KUKA KRL program: EPS_2_26115_ST7258_A_20260223020030.src

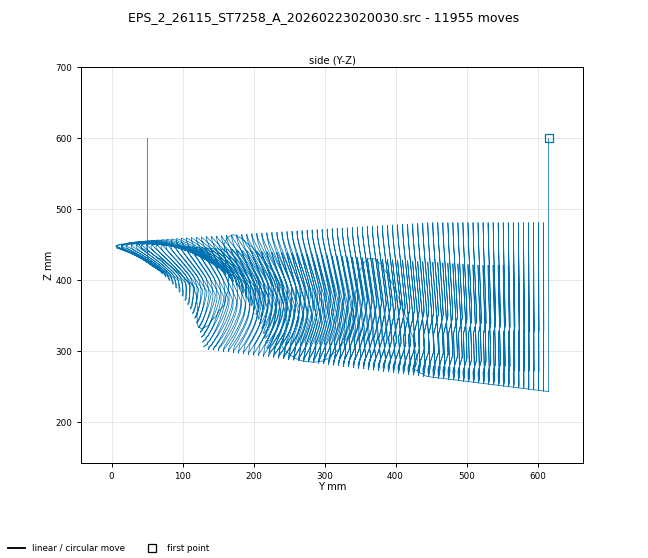
[picture p0: tool path of EPS_2_26115_ST7258_A_20260223020030.src, 11955 of 11957 moves have a stored position in this frame; points joined in program order, loops and branches not executed]
&ACCESS RVP
&REL 4
&COMMENT QRS 19112012
&PARAM EDITMASK = *
DEF PART()
EXT BAS (BAS_COMMAND :IN,REAL :IN )
INT I
BAS (#INITMOV,0 )

;KUKA QRS Post kuka4.cps  Date:22-06-2017 !

File_ID=3071

QRS_PRE_INIT()

;Init var - Until changes are made in qrs_pre_init
Outlet_Square_prg=0
Inlet_1_Square_prg=0
Inlet_2_Square_prg=0
Inlet_3_Square_prg=0
Inlet_4_Square_prg=0
Inlet_5_Square_prg=0

Outlet_1={X 0.000, Y 450.000, Z 332.000, B 0.000, E1 0.000 }
Inlet_1={X 0.000, Y 518.350, Z 272.000, B 0.000, E1 213.000 }
Outlet_1_type=299
Inlet_1_type=299
;QRS#1=Sidecore dimensions
;QRS#2=300-12" PVC SDR 35 Cut Back
;QRS#3=300-12" PVC SDR 35
;QRS#4=
;QRS#5=
;QRS#6=
;QRS#7=
;QRS#8=
;QRS#9=16M PSX
;QRS#10=16M PSX
;QRS#11=
;QRS#12=
;QRS#13=
;QRS#14=
;QRS#15=
;QRS#16=1220x127x762 2,5'
;QRS#17=EPS Height
;QRS#18=481,5
;QRS#19=*
;QRS#20= UPDATED VERSION 22-06-2017
;QRS#21=*
Outlet_Square=0150
Inlet_1_Square=0150
Inlet_2_Square=0
Inlet_3_Square=0
Inlet_4_Square=0
Inlet_5_Square=0
Mill_Square=1
Outlet_Square_Prg=216
Inlet_1_Square_prg=206

QRS_INIT()

$ADVANCE=5

; T1
PTP {E1 173.608,E2 173.608}
PTP {X 0,Y 615.508,A -85,B 0,C 180,E1 173.608,E2 173.608,E3 0,E4 0,E5 0,E6 0}
QRS_SPEED_INIT()
LIN {X 0,Y 615.508,Z 600,A -85,B 0,C 180,E1 173.608,E2 173.608,E3 0,E4 0,E5 0,E6 0} C_VEL
LIN {X 0,Y 615.508,Z 253.5,A -85,B 0,C 180,E1 173.608,E2 173.608} C_VEL
LIN {X 0,Y 615.508,Z 245.325,A -85,B 0,C 180,E1 173.608,E2 173.608} C_VEL
LIN {X 0,Y 615.49,Z 243.325,A -85,B 0,C 180,E1 173.422,E2 173.422} C_VEL
LIN {X 0,Y 615.476,Z 243.325,A -85,B 0,C 180,E1 170.802,E2 170.802} C_VEL
LIN {X 0,Y 615.493,Z 243.324,A -85,B 0,C 180,E1 168.14,E2 168.14} C_VEL
LIN {X 0,Y 615.493,Z 243.322,A -85,B 0,C 180,E1 165.452,E2 165.452} C_VEL
LIN {X 0,Y 615.477,Z 243.325,A -85,B 0,C 180,E1 162.73,E2 162.73} C_VEL
LIN {X 0,Y 615.492,Z 243.326,A -85,B 0,C 180,E1 159.968,E2 159.968} C_VEL
LIN {X 0,Y 615.478,Z 243.325,A -85,B 0,C 180,E1 157.156,E2 157.156} C_VEL
LIN {X 0,Y 615.487,Z 243.323,A -85,B 0,C 180,E1 154.432,E2 154.432} C_VEL
LIN {X 0,Y 615.497,Z 243.325,A -85,B 0,C 180,E1 151.549,E2 151.549} C_VEL
LIN {X 0,Y 615.474,Z 243.325,A -85,B 0,C 180,E1 148.917,E2 148.917} C_VEL
LIN {X 0,Y 615.486,Z 243.326,A -85,B 0,C 180,E1 146.467,E2 146.467} C_VEL
LIN {X 0,Y 615.483,Z 243.324,A -85,B 0,C 180,E1 143.576,E2 143.576} C_VEL
LIN {X 0,Y 615.486,Z 243.325,A -85,B 0,C 180,E1 140.939,E2 140.939} C_VEL
LIN {X 0,Y 615.491,Z 243.326,A -85,B 0,C 180,E1 137.92,E2 137.92} C_VEL
LIN {X 0,Y 615.49,Z 243.326,A -85,B 0,C 180,E1 134.933,E2 134.933} C_VEL
LIN {X 0,Y 615.49,Z 243.322,A -85,B 0,C 180,E1 132.082,E2 132.082} C_VEL
LIN {X 0,Y 615.489,Z 243.325,A -85,B 0,C 180,E1 129.75,E2 129.75} C_VEL
LIN {X 0,Y 615.475,Z 243.325,A -85,B 0,C 180,E1 126.937,E2 126.937} C_VEL
LIN {X 0,Y 615.481,Z 243.325,A -85,B 0,C 180,E1 124.702,E2 124.702} C_VEL
LIN {X 0,Y 615.497,Z 243.325,A -85,B 0,C 180,E1 122.335,E2 122.335} C_VEL
LIN {X 0,Y 615.477,Z 243.326,A -85,B 0,C 180,E1 119.407,E2 119.407} C_VEL
LIN {X 0,Y 615.498,Z 243.325,A -85,B 0,C 180,E1 117.05,E2 117.05} C_VEL
LIN {X 0,Y 615.492,Z 243.326,A -85,B 0,C 180,E1 114.012,E2 114.012} C_VEL
LIN {X 0,Y 615.475,Z 243.325,A -85,B 0,C 180,E1 111.433,E2 111.433} C_VEL
LIN {X 0,Y 615.488,Z 243.326,A -85,B 0,C 180,E1 108.609,E2 108.609} C_VEL
LIN {X 0,Y 615.478,Z 243.325,A -85,B 0,C 180,E1 105.906,E2 105.906} C_VEL
LIN {X 0,Y 615.485,Z 243.324,A -85,B 0,C 180,E1 103.202,E2 103.202} C_VEL
LIN {X 0,Y 615.495,Z 243.323,A -85,B 0,C 180,E1 100.527,E2 100.527} C_VEL
LIN {X 0,Y 615.476,Z 243.325,A -85,B 0,C 180,E1 97.876,E2 97.876} C_VEL
LIN {X 0,Y 615.488,Z 243.326,A -85,B 0,C 180,E1 95.242,E2 95.242} C_VEL
LIN {X 0,Y 615.479,Z 246.1,A -85,B 0,C 180,E1 92.618,E2 92.618} C_VEL
LIN {X 0,Y 615.467,Z 248.837,A -85,B 0,C 180,E1 90,E2 90} C_VEL
LIN {X 0,Y 615.457,Z 251.727,A -85,B 0,C 180,E1 87.382,E2 87.382} C_VEL
LIN {X 0,Y 615.479,Z 254.78,A -85,B 0,C 180,E1 84.759,E2 84.759} C_VEL
LIN {X 0,Y 615.427,Z 257.933,A -85,B 0,C 180,E1 82.124,E2 82.124} C_VEL
LIN {X 0,Y 615.459,Z 261.171,A -85,B 0,C 180,E1 79.473,E2 79.473} C_VEL
LIN {X 0,Y 615.457,Z 264.49,A -85,B 0,C 180,E1 76.799,E2 76.799} C_VEL
LIN {X 0,Y 615.42,Z 267.919,A -85,B 0,C 180,E1 74.094,E2 74.094} C_VEL
LIN {X 0,Y 615.488,Z 268.917,A -85,B 0,C 180,E1 73.307,E2 73.307} C_VEL
LIN {X 0,Y 615.462,Z 288.21,A -85,B 0,C 180,E1 72.943,E2 72.943} C_VEL
LIN {X 0,Y 615.424,Z 303.447,A -85,B 0,C 180,E1 72.514,E2 72.514} C_VEL
LIN {X 0,Y 615.425,Z 318.039,A -85,B 0,C 180,E1 71.961,E2 71.961} C_VEL
LIN {X 0,Y 615.488,Z 332.329,A -85,B 0,C 180,E1 71.268,E2 71.268} C_VEL
LIN {X 0,Y 615.5,Z 345.387,A -85,B 0,C 180,E1 70.49,E2 70.49} C_VEL
LIN {X 0,Y 615.497,Z 358.126,A -85,B 0,C 180,E1 69.57,E2 69.57} C_VEL
LIN {X 0,Y 615.496,Z 369.68,A -85,B 0,C 180,E1 68.569,E2 68.569} C_VEL
LIN {X 0,Y 615.497,Z 379.793,A -85,B 0,C 180,E1 67.526,E2 67.526} C_VEL
LIN {X 0,Y 615.494,Z 388.648,A -85,B 0,C 180,E1 66.445,E2 66.445} C_VEL
LIN {X 0,Y 615.495,Z 397.207,A -85,B 0,C 180,E1 65.189,E2 65.189} C_VEL
LIN {X 0,Y 615.492,Z 404.275,A -85,B 0,C 180,E1 63.921,E2 63.921} C_VEL
LIN {X 0,Y 615.492,Z 409.272,A -85,B 0,C 180,E1 62.824,E2 62.824} C_VEL
LIN {X 0,Y 615.496,Z 413.84,A -85,B 0,C 180,E1 61.546,E2 61.546} C_VEL
LIN {X 0,Y 615.494,Z 417.375,A -85,B 0,C 180,E1 60.202,E2 60.202} C_VEL
LIN {X 0,Y 615.492,Z 419.603,A -85,B 0,C 180,E1 58.911,E2 58.911} C_VEL
LIN {X 0,Y 615.496,Z 420.755,A -85,B 0,C 180,E1 57.544,E2 57.544} C_VEL
LIN {X 0,Y 615.491,Z 420.778,A -85,B 0,C 180,E1 56.463,E2 56.463} C_VEL
LIN {X 0,Y 615.495,Z 419.823,A -85,B 0,C 180,E1 55.186,E2 55.186} C_VEL
LIN {X 0,Y 615.491,Z 418.313,A -85,B 0,C 180,E1 54.164,E2 54.164} C_VEL
LIN {X 0,Y 615.492,Z 415.024,A -85,B 0,C 180,E1 52.759,E2 52.759} C_VEL
LIN {X 0,Y 615.496,Z 410.925,A -85,B 0,C 180,E1 51.516,E2 51.516} C_VEL
LIN {X 0,Y 615.496,Z 405.553,A -85,B 0,C 180,E1 50.251,E2 50.251} C_VEL
LIN {X 0,Y 615.493,Z 398.318,A -85,B 0,C 180,E1 48.903,E2 48.903} C_VEL
LIN {X 0,Y 615.5,Z 390.008,A -85,B 0,C 180,E1 47.649,E2 47.649} C_VEL
LIN {X 0,Y 615.494,Z 381.434,A -85,B 0,C 180,E1 46.568,E2 46.568} C_VEL
LIN {X 0,Y 615.499,Z 370.947,A -85,B 0,C 180,E1 45.461,E2 45.461} C_VEL
LIN {X 0,Y 615.494,Z 359.396,A -85,B 0,C 180,E1 44.441,E2 44.441} C_VEL
LIN {X 0,Y 615.493,Z 346.979,A -85,B 0,C 180,E1 43.525,E2 43.525} C_VEL
LIN {X 0,Y 615.495,Z 333.385,A -85,B 0,C 180,E1 42.699,E2 42.699} C_VEL
LIN {X 0,Y 615.485,Z 321.059,A -85,B 0,C 180,E1 42.081,E2 42.081} C_VEL
LIN {X 0,Y 615.478,Z 306.886,A -85,B 0,C 180,E1 41.511,E2 41.511} C_VEL
LIN {X 0,Y 615.477,Z 291.025,A -85,B 0,C 180,E1 41.033,E2 41.033} C_VEL
LIN {X 0,Y 615.482,Z 275.439,A -85,B 0,C 180,E1 40.712,E2 40.712} C_VEL
LIN {X 0,Y 615.485,Z 268.921,A -85,B 0,C 180,E1 40.605,E2 40.605} C_VEL
LIN {X 0,Y 615.484,Z 265.619,A -85,B 0,C 180,E1 38.013,E2 38.013} C_VEL
LIN {X 0,Y 615.479,Z 262.614,A -85,B 0,C 180,E1 35.615,E2 35.615} C_VEL
LIN {X 0,Y 615.48,Z 259.684,A -85,B 0,C 180,E1 33.235,E2 33.235} C_VEL
LIN {X 0,Y 615.487,Z 256.886,A -85,B 0,C 180,E1 30.918,E2 30.918} C_VEL
LIN {X 0,Y 615.477,Z 253.956,A -85,B 0,C 180,E1 28.45,E2 28.45} C_VEL
LIN {X 0,Y 615.481,Z 250.784,A -85,B 0,C 180,E1 25.715,E2 25.715} C_VEL
LIN {X 0,Y 615.487,Z 248.533,A -85,B 0,C 180,E1 23.555,E2 23.555} C_VEL
LIN {X 0,Y 615.456,Z 246.383,A -85,B 0,C 180,E1 21.432,E2 21.432} C_VEL
LIN {X 0,Y 615.496,Z 243.418,A -85,B 0,C 180,E1 18.609,E2 18.609} C_VEL
LIN {X 0,Y 615.486,Z 243.323,A -85,B 0,C 180,E1 15.904,E2 15.904} C_VEL
LIN {X 0,Y 615.487,Z 243.325,A -85,B 0,C 180,E1 13.2,E2 13.2} C_VEL
LIN {X 0,Y 615.487,Z 243.323,A -85,B 0,C 180,E1 10.526,E2 10.526} C_VEL
LIN {X 0,Y 615.484,Z 243.325,A -85,B 0,C 180,E1 7.875,E2 7.875} C_VEL
LIN {X 0,Y 615.478,Z 243.325,A -85,B 0,C 180,E1 5.241,E2 5.241} C_VEL
LIN {X 0,Y 615.496,Z 243.323,A -85,B 0,C 180,E1 2.617,E2 2.617} C_VEL
LIN {X 0,Y 615.483,Z 243.324,A -85,B 0,C 180,E1 -0.001,E2 -0.001} C_VEL
LIN {X 0,Y 615.49,Z 243.325,A -85,B 0,C 180,E1 -2.619,E2 -2.619} C_VEL
LIN {X 0,Y 615.49,Z 243.322,A -85,B 0,C 180,E1 -5.242,E2 -5.242} C_VEL
LIN {X 0,Y 615.484,Z 243.326,A -85,B 0,C 180,E1 -7.876,E2 -7.876} C_VEL
LIN {X 0,Y 615.474,Z 243.325,A -85,B 0,C 180,E1 -10.528,E2 -10.528} C_VEL
LIN {X 0,Y 615.498,Z 243.323,A -85,B 0,C 180,E1 -13.202,E2 -13.202} C_VEL
LIN {X 0,Y 615.481,Z 243.324,A -85,B 0,C 180,E1 -15.906,E2 -15.906} C_VEL
LIN {X 0,Y 615.48,Z 243.325,A -85,B 0,C 180,E1 -18.647,E2 -18.647} C_VEL
LIN {X 0,Y 615.498,Z 243.324,A -85,B 0,C 180,E1 -21.432,E2 -21.432} C_VEL
LIN {X 0,Y 615.473,Z 243.326,A -85,B 0,C 180,E1 -24.273,E2 -24.273} C_VEL
LIN {X 0,Y 615.498,Z 243.321,A -85,B 0,C 180,E1 -27.048,E2 -27.048} C_VEL
LIN {X 0,Y 615.49,Z 243.325,A -85,B 0,C 180,E1 -29.796,E2 -29.796} C_VEL
LIN {X 0,Y 615.481,Z 243.324,A -85,B 0,C 180,E1 -32.458,E2 -32.458} C_VEL
LIN {X 0,Y 615.493,Z 243.321,A -85,B 0,C 180,E1 -34.815,E2 -34.815} C_VEL
LIN {X 0,Y 615.491,Z 243.325,A -85,B 0,C 180,E1 -37.242,E2 -37.242} C_VEL
LIN {X 0,Y 615.474,Z 243.325,A -85,B 0,C 180,E1 -40.088,E2 -40.088} C_VEL
LIN {X 0,Y 615.481,Z 243.325,A -85,B 0,C 180,E1 -42.354,E2 -42.354} C_VEL
LIN {X 0,Y 615.478,Z 243.325,A -85,B 0,C 180,E1 -45.07,E2 -45.07} C_VEL
LIN {X 0,Y 615.497,Z 243.325,A -85,B 0,C 180,E1 -47.919,E2 -47.919} C_VEL
LIN {X 0,Y 615.498,Z 243.517,A -85,B 0,C 180,E1 -48.717,E2 -48.717} C_VEL
LIN {X 0,Y 615.467,Z 250.403,A -85,B 0,C 180,E1 -51.095,E2 -51.095} C_VEL
LIN {X 0,Y 615.424,Z 257.825,A -85,B 0,C 180,E1 -53.572,E2 -53.572} C_VEL
LIN {X 0,Y 615.43,Z 265.245,A -85,B 0,C 180,E1 -55.975,E2 -55.975} C_VEL
LIN {X 0,Y 615.47,Z 272.654,A -85,B 0,C 180,E1 -58.314,E2 -58.314} C_VEL
LIN {X 0,Y 615.44,Z 281.3,A -85,B 0,C 180,E1 -60.967,E2 -60.967} C_VEL
LIN {X 0,Y 615.44,Z 287.95,A -85,B 0,C 180,E1 -62.964,E2 -62.964} C_VEL
LIN {X 0,Y 615.439,Z 294.876,A -85,B 0,C 180,E1 -65.007,E2 -65.007} C_VEL
LIN {X 0,Y 615.436,Z 302.279,A -85,B 0,C 180,E1 -67.154,E2 -67.154} C_VEL
LIN {X 0,Y 615.448,Z 310.326,A -85,B 0,C 180,E1 -69.453,E2 -69.453} C_VEL
LIN {X 0,Y 615.487,Z 320.751,A -85,B 0,C 180,E1 -72.387,E2 -72.387} C_VEL
LIN {X 0,Y 615.477,Z 325.142,A -85,B 0,C 180,E1 -73.606,E2 -73.606} C_VEL
LIN {X 0,Y 615.494,Z 343.255,A -85,B 0,C 180,E1 -73.9,E2 -73.9} C_VEL
LIN {X 0,Y 615.497,Z 357.822,A -85,B 0,C 180,E1 -74.266,E2 -74.266} C_VEL
LIN {X 0,Y 615.456,Z 372.682,A -85,B 0,C 180,E1 -74.774,E2 -74.774} C_VEL
LIN {X 0,Y 615.465,Z 386.117,A -85,B 0,C 180,E1 -75.366,E2 -75.366} C_VEL
LIN {X 0,Y 615.498,Z 400.019,A -85,B 0,C 180,E1 -76.127,E2 -76.127} C_VEL
LIN {X 0,Y 615.496,Z 412.639,A -85,B 0,C 180,E1 -76.967,E2 -76.967} C_VEL
LIN {X 0,Y 615.496,Z 423.235,A -85,B 0,C 180,E1 -77.805,E2 -77.805} C_VEL
LIN {X 0,Y 615.496,Z 433.979,A -85,B 0,C 180,E1 -78.808,E2 -78.808} C_VEL
LIN {X 0,Y 615.496,Z 444.426,A -85,B 0,C 180,E1 -79.972,E2 -79.972} C_VEL
LIN {X 0,Y 615.495,Z 453.105,A -85,B 0,C 180,E1 -81.133,E2 -81.133} C_VEL
LIN {X 0,Y 615.493,Z 461.227,A -85,B 0,C 180,E1 -82.455,E2 -82.455} C_VEL
LIN {X 0,Y 615.496,Z 467.731,A -85,B 0,C 180,E1 -83.773,E2 -83.773} C_VEL
LIN {X 0,Y 615.496,Z 472.81,A -85,B 0,C 180,E1 -85.088,E2 -85.088} C_VEL
LIN {X 0,Y 615.495,Z 475.741,A -85,B 0,C 180,E1 -86.072,E2 -86.072} C_VEL
LIN {X 0,Y 615.494,Z 478.601,A -85,B 0,C 180,E1 -87.383,E2 -87.383} C_VEL
LIN {X 0,Y 615.492,Z 480.307,A -85,B 0,C 180,E1 -88.692,E2 -88.692} C_VEL
LIN {X 0,Y 615.491,Z 480.889,A -85,B 0,C 180,E1 -90,E2 -90} C_VEL
LIN {X 0,Y 615.492,Z 480.306,A -85,B 0,C 180,E1 -91.309,E2 -91.309} C_VEL
LIN {X 0,Y 615.494,Z 478.599,A -85,B 0,C 180,E1 -92.618,E2 -92.618} C_VEL
LIN {X 0,Y 615.495,Z 475.739,A -85,B 0,C 180,E1 -93.929,E2 -93.929} C_VEL
LIN {X 0,Y 615.491,Z 471.664,A -85,B 0,C 180,E1 -95.242,E2 -95.242} C_VEL
LIN {X 0,Y 615.49,Z 466.16,A -85,B 0,C 180,E1 -96.58,E2 -96.58} C_VEL
LIN {X 0,Y 615.493,Z 459.39,A -85,B 0,C 180,E1 -97.876,E2 -97.876} C_VEL
LIN {X 0,Y 615.495,Z 450.806,A -85,B 0,C 180,E1 -99.199,E2 -99.199} C_VEL
LIN {X 0,Y 615.494,Z 441.663,A -85,B 0,C 180,E1 -100.361,E2 -100.361} C_VEL
LIN {X 0,Y 615.497,Z 432.35,A -85,B 0,C 180,E1 -101.36,E2 -101.36} C_VEL
LIN {X 0,Y 615.496,Z 421.288,A -85,B 0,C 180,E1 -102.363,E2 -102.363} C_VEL
LIN {X 0,Y 615.498,Z 409.147,A -85,B 0,C 180,E1 -103.285,E2 -103.285} C_VEL
LIN {X 0,Y 615.498,Z 396.405,A -85,B 0,C 180,E1 -104.09,E2 -104.09} C_VEL
LIN {X 0,Y 615.456,Z 382.602,A -85,B 0,C 180,E1 -104.804,E2 -104.804} C_VEL
LIN {X 0,Y 615.465,Z 368.172,A -85,B 0,C 180,E1 -105.397,E2 -105.397} C_VEL
LIN {X 0,Y 615.494,Z 353.234,A -85,B 0,C 180,E1 -105.863,E2 -105.863} C_VEL
LIN {X 0,Y 615.493,Z 337.989,A -85,B 0,C 180,E1 -106.198,E2 -106.198} C_VEL
LIN {X 0,Y 615.477,Z 325.142,A -85,B 0,C 180,E1 -106.394,E2 -106.394} C_VEL
LIN {X 0,Y 615.445,Z 315.833,A -85,B 0,C 180,E1 -108.993,E2 -108.993} C_VEL
LIN {X 0,Y 615.497,Z 305.962,A -85,B 0,C 180,E1 -111.784,E2 -111.784} C_VEL
LIN {X 0,Y 615.449,Z 297.34,A -85,B 0,C 180,E1 -114.274,E2 -114.274} C_VEL
LIN {X 0,Y 615.431,Z 289.943,A -85,B 0,C 180,E1 -116.447,E2 -116.447} C_VEL
LIN {X 0,Y 615.422,Z 282.534,A -85,B 0,C 180,E1 -118.662,E2 -118.662} C_VEL
LIN {X 0,Y 615.445,Z 274.614,A -85,B 0,C 180,E1 -121.079,E2 -121.079} C_VEL
LIN {X 0,Y 615.485,Z 266.771,A -85,B 0,C 180,E1 -123.534,E2 -123.534} C_VEL
LIN {X 0,Y 615.446,Z 259.654,A -85,B 0,C 180,E1 -125.828,E2 -125.828} C_VEL
LIN {X 0,Y 615.431,Z 252.875,A -85,B 0,C 180,E1 -128.073,E2 -128.073} C_VEL
LIN {X 0,Y 615.432,Z 246.975,A -85,B 0,C 180,E1 -130.083,E2 -130.083} C_VEL
LIN {X 0,Y 615.495,Z 243.321,A -85,B 0,C 180,E1 -131.379,E2 -131.379} C_VEL
LIN {X 0,Y 615.497,Z 243.325,A -85,B 0,C 180,E1 -134.149,E2 -134.149} C_VEL
LIN {X 0,Y 615.484,Z 243.323,A -85,B 0,C 180,E1 -136.953,E2 -136.953} C_VEL
LIN {X 0,Y 615.492,Z 243.326,A -85,B 0,C 180,E1 -139.394,E2 -139.394} C_VEL
LIN {X 0,Y 615.474,Z 243.325,A -85,B 0,C 180,E1 -141.99,E2 -141.99} C_VEL
LIN {X 0,Y 615.481,Z 243.325,A -85,B 0,C 180,E1 -144.383,E2 -144.383} C_VEL
LIN {X 0,Y 615.492,Z 243.326,A -85,B 0,C 180,E1 -146.764,E2 -146.764} C_VEL
LIN {X 0,Y 615.491,Z 243.323,A -85,B 0,C 180,E1 -149.08,E2 -149.08} C_VEL
LIN {X 0,Y 615.478,Z 243.324,A -85,B 0,C 180,E1 -151.552,E2 -151.552} C_VEL
LIN {X 0,Y 615.486,Z 243.324,A -85,B 0,C 180,E1 -154.284,E2 -154.284} C_VEL
LIN {X 0,Y 615.494,Z 243.326,A -85,B 0,C 180,E1 -157.155,E2 -157.155} C_VEL
LIN {X 0,Y 615.477,Z 243.325,A -85,B 0,C 180,E1 -159.966,E2 -159.966} C_VEL
LIN {X 0,Y 615.496,Z 243.321,A -85,B 0,C 180,E1 -162.729,E2 -162.729} C_VEL
LIN {X 0,Y 615.494,Z 243.324,A -85,B 0,C 180,E1 -165.451,E2 -165.451} C_VEL
LIN {X 0,Y 615.475,Z 243.325,A -85,B 0,C 180,E1 -168.138,E2 -168.138} C_VEL
LIN {X 0,Y 615.497,Z 243.325,A -85,B 0,C 180,E1 -170.801,E2 -170.801} C_VEL
LIN {X 0,Y 615.475,Z 243.325,A -85,B 0,C 180,E1 -173.443,E2 -173.443} C_VEL
LIN {X 0,Y 615.491,Z 243.326,A -85,B 0,C 180,E1 -176.071,E2 -176.071} C_VEL
LIN {X 0,Y 615.493,Z 243.321,A -85,B 0,C 180,E1 -178.691,E2 -178.691} C_VEL
LIN {X 0,Y 615.489,Z 243.326,A -85,B 0,C 180,E1 -181.308,E2 -181.308} C_VEL
LIN {X 0,Y 615.475,Z 243.325,A -85,B 0,C 180,E1 -183.928,E2 -183.928} C_VEL
LIN {X 0,Y 615.49,Z 243.325,A -85,B 0,C 180,E1 -186.578,E2 -186.578} C_VEL
LIN {X 0,Y 614.807,Z 243.471,A -85,B 0,C 180,E1 -187.124,E2 -187.124} C_VEL
LIN {X 0,Y 611.965,Z 243.883,A -85,B 0,C 180,E1 -188.01,E2 -188.01} C_VEL
LIN {X 0,Y 609.573,Z 244.193,A -85,B 0,C 180,E1 -188.722,E2 -188.722} C_VEL
LIN {X 0,Y 608.541,Z 244.311,A -85,B 0,C 180,E1 -189.272,E2 -189.272} C_VEL
LIN {X 0,Y 608.453,Z 244.32,A -85,B 0,C 180,E1 -189.458,E2 -189.458} C_VEL
LIN {X 0,Y 608.468,Z 244.319,A -85,B 0,C 180,E1 -191.999,E2 -191.999} C_VEL
LIN {X 0,Y 608.476,Z 244.319,A -85,B 0,C 180,E1 -194.72,E2 -194.72} C_VEL
LIN {X 0,Y 608.45,Z 244.321,A -85,B 0,C 180,E1 -197.476,E2 -197.476} C_VEL
LIN {X 0,Y 608.461,Z 244.32,A -85,B 0,C 180,E1 -200.273,E2 -200.273} C_VEL
LIN {X 0,Y 608.459,Z 244.32,A -85,B 0,C 180,E1 -202.475,E2 -202.475} C_VEL
LIN {X 0,Y 608.454,Z 244.321,A -85,B 0,C 180,E1 -204.57,E2 -204.57} C_VEL
LIN {X 0,Y 608.474,Z 244.319,A -85,B 0,C 180,E1 -207.206,E2 -207.206} C_VEL
LIN {X 0,Y 608.472,Z 244.318,A -85,B 0,C 180,E1 -209.972,E2 -209.972} C_VEL
LIN {X 0,Y 608.454,Z 244.321,A -85,B 0,C 180,E1 -212.878,E2 -212.878} C_VEL
LIN {X 0,Y 608.446,Z 244.321,A -85,B 0,C 180,E1 -215.276,E2 -215.276} C_VEL
LIN {X 0,Y 608.465,Z 244.319,A -85,B 0,C 180,E1 -218.24,E2 -218.24} C_VEL
LIN {X 0,Y 608.445,Z 244.321,A -85,B 0,C 180,E1 -220.328,E2 -220.328} C_VEL
LIN {X 0,Y 608.453,Z 244.322,A -85,B 0,C 180,E1 -222.958,E2 -222.958} C_VEL
LIN {X 0,Y 608.463,Z 244.319,A -85,B 0,C 180,E1 -225.734,E2 -225.734} C_VEL
LIN {X 0,Y 608.455,Z 244.32,A -85,B 0,C 180,E1 -228.657,E2 -228.657} C_VEL
LIN {X 0,Y 608.463,Z 244.322,A -85,B 0,C 180,E1 -231.411,E2 -231.411} C_VEL
LIN {X 0,Y 608.471,Z 244.318,A -85,B 0,C 180,E1 -233.949,E2 -233.949} C_VEL
LIN {X 0,Y 608.458,Z 244.32,A -85,B 0,C 180,E1 -236.328,E2 -236.328} C_VEL
LIN {X 0,Y 608.472,Z 244.321,A -85,B 0,C 180,E1 -238.726,E2 -238.726} C_VEL
LIN {X 0,Y 608.476,Z 244.317,A -85,B 0,C 180,E1 -241.377,E2 -241.377} C_VEL
LIN {X 0,Y 608.443,Z 244.324,A -85,B 0,C 180,E1 -243.964,E2 -243.964} C_VEL
LIN {X 0,Y 608.467,Z 244.32,A -85,B 0,C 180,E1 -246.155,E2 -246.155} C_VEL
LIN {X 0,Y 608.455,Z 244.321,A -85,B 0,C 180,E1 -249.018,E2 -249.018} C_VEL
LIN {X 0,Y 608.445,Z 244.321,A -85,B 0,C 180,E1 -251.828,E2 -251.828} C_VEL
LIN {X 0,Y 608.467,Z 244.32,A -85,B 0,C 180,E1 -254.594,E2 -254.594} C_VEL
LIN {X 0,Y 608.478,Z 244.318,A -85,B 0,C 180,E1 -257.323,E2 -257.323} C_VEL
LIN {X 0,Y 608.448,Z 244.321,A -85,B 0,C 180,E1 -260.022,E2 -260.022} C_VEL
LIN {X 0,Y 608.481,Z 244.319,A -85,B 0,C 180,E1 -262.7,E2 -262.7} C_VEL
LIN {X 0,Y 608.466,Z 244.32,A -85,B 0,C 180,E1 -264.698,E2 -264.698} C_VEL
LIN {X 0,Y 608.446,Z 246.912,A -85,B 0,C 180,E1 -267.351,E2 -267.351} C_VEL
LIN {X 0,Y 608.416,Z 249.67,A -85,B 0,C 180,E1 -270,E2 -270} C_VEL
LIN {X 0,Y 608.398,Z 252.528,A -85,B 0,C 180,E1 -272.648,E2 -272.648} C_VEL
LIN {X 0,Y 608.436,Z 255.607,A -85,B 0,C 180,E1 -275.302,E2 -275.302} C_VEL
LIN {X 0,Y 608.369,Z 258.782,A -85,B 0,C 180,E1 -277.968,E2 -277.968} C_VEL
LIN {X 0,Y 608.41,Z 262.041,A -85,B 0,C 180,E1 -280.65,E2 -280.65} C_VEL
LIN {X 0,Y 608.392,Z 265.398,A -85,B 0,C 180,E1 -283.358,E2 -283.358} C_VEL
LIN {X 0,Y 608.374,Z 268.851,A -85,B 0,C 180,E1 -286.096,E2 -286.096} C_VEL
LIN {X 0,Y 608.431,Z 269.427,A -85,B 0,C 180,E1 -286.522,E2 -286.522} C_VEL
LIN {X 0,Y 608.668,Z 276.786,A -85,B 0,C 180,E1 -286.637,E2 -286.637} C_VEL
LIN {X 0,Y 608.606,Z 292.383,A -85,B 0,C 180,E1 -286.974,E2 -286.974} C_VEL
LIN {X 0,Y 608.563,Z 307.119,A -85,B 0,C 180,E1 -287.429,E2 -287.429} C_VEL
LIN {X 0,Y 608.534,Z 321.01,A -85,B 0,C 180,E1 -287.995,E2 -287.995} C_VEL
LIN {X 0,Y 608.576,Z 335.698,A -85,B 0,C 180,E1 -288.749,E2 -288.749} C_VEL
LIN {X 0,Y 608.558,Z 348.631,A -85,B 0,C 180,E1 -289.567,E2 -289.567} C_VEL
LIN {X 0,Y 608.52,Z 361.411,A -85,B 0,C 180,E1 -290.54,E2 -290.54} C_VEL
LIN {X 0,Y 608.481,Z 372.102,A -85,B 0,C 180,E1 -291.513,E2 -291.513} C_VEL
LIN {X 0,Y 608.478,Z 381.894,A -85,B 0,C 180,E1 -292.566,E2 -292.566} C_VEL
LIN {X 0,Y 608.479,Z 391.857,A -85,B 0,C 180,E1 -293.844,E2 -293.844} C_VEL
LIN {X 0,Y 608.452,Z 399.992,A -85,B 0,C 180,E1 -295.118,E2 -295.118} C_VEL
LIN {X 0,Y 608.454,Z 406.66,A -85,B 0,C 180,E1 -296.403,E2 -296.403} C_VEL
LIN {X 0,Y 608.434,Z 411.324,A -85,B 0,C 180,E1 -297.518,E2 -297.518} C_VEL
LIN {X 0,Y 608.424,Z 415.044,A -85,B 0,C 180,E1 -298.614,E2 -298.614} C_VEL
LIN {X 0,Y 608.419,Z 418.388,A -85,B 0,C 180,E1 -299.966,E2 -299.966} C_VEL
LIN {X 0,Y 608.413,Z 420.498,A -85,B 0,C 180,E1 -301.319,E2 -301.319} C_VEL
LIN {X 0,Y 608.419,Z 421.382,A -85,B 0,C 180,E1 -302.518,E2 -302.518} C_VEL
LIN {X 0,Y 608.417,Z 421.345,A -85,B 0,C 180,E1 -303.729,E2 -303.729} C_VEL
LIN {X 0,Y 608.419,Z 420.341,A -85,B 0,C 180,E1 -304.904,E2 -304.904} C_VEL
LIN {X 0,Y 608.442,Z 418.457,A -85,B 0,C 180,E1 -306.092,E2 -306.092} C_VEL
LIN {X 0,Y 608.43,Z 415.923,A -85,B 0,C 180,E1 -307.156,E2 -307.156} C_VEL
LIN {X 0,Y 608.427,Z 411.256,A -85,B 0,C 180,E1 -308.59,E2 -308.59} C_VEL
LIN {X 0,Y 608.436,Z 405.765,A -85,B 0,C 180,E1 -309.871,E2 -309.871} C_VEL
LIN {X 0,Y 608.439,Z 398.755,A -85,B 0,C 180,E1 -311.177,E2 -311.177} C_VEL
LIN {X 0,Y 608.473,Z 390.369,A -85,B 0,C 180,E1 -312.449,E2 -312.449} C_VEL
LIN {X 0,Y 608.473,Z 381.58,A -85,B 0,C 180,E1 -313.56,E2 -313.56} C_VEL
LIN {X 0,Y 608.491,Z 371.388,A -85,B 0,C 180,E1 -314.645,E2 -314.645} C_VEL
LIN {X 0,Y 608.507,Z 360.192,A -85,B 0,C 180,E1 -315.649,E2 -315.649} C_VEL
LIN {X 0,Y 608.547,Z 347.477,A -85,B 0,C 180,E1 -316.601,E2 -316.601} C_VEL
LIN {X 0,Y 608.586,Z 334.717,A -85,B 0,C 180,E1 -317.394,E2 -317.394} C_VEL
LIN {X 0,Y 608.597,Z 320.908,A -85,B 0,C 180,E1 -318.098,E2 -318.098} C_VEL
LIN {X 0,Y 608.611,Z 306.371,A -85,B 0,C 180,E1 -318.686,E2 -318.686} C_VEL
LIN {X 0,Y 608.639,Z 290.791,A -85,B 0,C 180,E1 -319.157,E2 -319.157} C_VEL
LIN {X 0,Y 608.672,Z 275.607,A -85,B 0,C 180,E1 -319.473,E2 -319.473} C_VEL
LIN {X 0,Y 608.552,Z 270.28,A -85,B 0,C 180,E1 -319.552,E2 -319.552} C_VEL
LIN {X 0,Y 608.426,Z 269.368,A -85,B 0,C 180,E1 -319.586,E2 -319.586} C_VEL
LIN {X 0,Y 608.413,Z 266,A -85,B 0,C 180,E1 -322.251,E2 -322.251} C_VEL
LIN {X 0,Y 608.408,Z 262.926,A -85,B 0,C 180,E1 -324.721,E2 -324.721} C_VEL
LIN {X 0,Y 608.418,Z 259.991,A -85,B 0,C 180,E1 -327.119,E2 -327.119} C_VEL
LIN {X 0,Y 608.45,Z 256.5,A -85,B 0,C 180,E1 -330.03,E2 -330.03} C_VEL
LIN {X 0,Y 608.431,Z 253.264,A -85,B 0,C 180,E1 -332.8,E2 -332.8} C_VEL
LIN {X 0,Y 608.453,Z 250.402,A -85,B 0,C 180,E1 -335.43,E2 -335.43} C_VEL
LIN {X 0,Y 608.429,Z 247.513,A -85,B 0,C 180,E1 -338.308,E2 -338.308} C_VEL
LIN {X 0,Y 608.434,Z 245.308,A -85,B 0,C 180,E1 -340.43,E2 -340.43} C_VEL
LIN {X 0,Y 608.454,Z 244.4,A -85,B 0,C 180,E1 -341.287,E2 -341.287} C_VEL
LIN {X 0,Y 608.462,Z 244.319,A -85,B 0,C 180,E1 -343.907,E2 -343.907} C_VEL
LIN {X 0,Y 608.463,Z 244.322,A -85,B 0,C 180,E1 -346.644,E2 -346.644} C_VEL
LIN {X 0,Y 608.463,Z 244.319,A -85,B 0,C 180,E1 -349.351,E2 -349.351} C_VEL
LIN {X 0,Y 608.476,Z 244.319,A -85,B 0,C 180,E1 -352.034,E2 -352.034} C_VEL
LIN {X 0,Y 608.459,Z 244.32,A -85,B 0,C 180,E1 -354.699,E2 -354.699} C_VEL
LIN {X 0,Y 608.485,Z 244.318,A -85,B 0,C 180,E1 -357.353,E2 -357.353} C_VEL
LIN {X 0,Y 608.474,Z 244.318,A -85,B 0,C 180,E1 -360.001,E2 -360.001} C_VEL
LIN {X 0,Y 608.48,Z 244.318,A -85,B 0,C 180,E1 -362.649,E2 -362.649} C_VEL
LIN {X 0,Y 608.468,Z 244.319,A -85,B 0,C 180,E1 -365.302,E2 -365.302} C_VEL
LIN {X 0,Y 608.475,Z 244.319,A -85,B 0,C 180,E1 -367.968,E2 -367.968} C_VEL
LIN {X 0,Y 608.458,Z 244.32,A -85,B 0,C 180,E1 -370.651,E2 -370.651} C_VEL
LIN {X 0,Y 608.472,Z 244.318,A -85,B 0,C 180,E1 -373.357,E2 -373.357} C_VEL
LIN {X 0,Y 608.457,Z 244.322,A -85,B 0,C 180,E1 -376.094,E2 -376.094} C_VEL
LIN {X 0,Y 608.454,Z 244.32,A -85,B 0,C 180,E1 -378.87,E2 -378.87} C_VEL
LIN {X 0,Y 608.471,Z 244.319,A -85,B 0,C 180,E1 -381.692,E2 -381.692} C_VEL
LIN {X 0,Y 608.451,Z 244.323,A -85,B 0,C 180,E1 -384.572,E2 -384.572} C_VEL
LIN {X 0,Y 608.485,Z 244.316,A -85,B 0,C 180,E1 -387.21,E2 -387.21} C_VEL
LIN {X 0,Y 608.468,Z 244.321,A -85,B 0,C 180,E1 -389.973,E2 -389.973} C_VEL
LIN {X 0,Y 608.455,Z 244.321,A -85,B 0,C 180,E1 -392.88,E2 -392.88} C_VEL
LIN {X 0,Y 608.437,Z 244.325,A -85,B 0,C 180,E1 -395.278,E2 -395.278} C_VEL
LIN {X 0,Y 608.465,Z 244.319,A -85,B 0,C 180,E1 -397.747,E2 -397.747} C_VEL
LIN {X 0,Y 608.449,Z 244.322,A -85,B 0,C 180,E1 -400.33,E2 -400.33} C_VEL
LIN {X 0,Y 608.47,Z 244.319,A -85,B 0,C 180,E1 -403.31,E2 -403.31} C_VEL
LIN {X 0,Y 608.471,Z 244.319,A -85,B 0,C 180,E1 -406.132,E2 -406.132} C_VEL
LIN {X 0,Y 608.469,Z 244.331,A -85,B 0,C 180,E1 -408.425,E2 -408.425} C_VEL
LIN {X 0,Y 608.524,Z 251.827,A -85,B 0,C 180,E1 -411.056,E2 -411.056} C_VEL
LIN {X 0,Y 608.47,Z 259.071,A -85,B 0,C 180,E1 -413.5,E2 -413.5} C_VEL
LIN {X 0,Y 608.453,Z 265.26,A -85,B 0,C 180,E1 -415.53,E2 -415.53} C_VEL
LIN {X 0,Y 608.446,Z 272.686,A -85,B 0,C 180,E1 -417.905,E2 -417.905} C_VEL
LIN {X 0,Y 608.502,Z 281.351,A -85,B 0,C 180,E1 -420.603,E2 -420.603} C_VEL
LIN {X 0,Y 608.418,Z 290.016,A -85,B 0,C 180,E1 -423.225,E2 -423.225} C_VEL
LIN {X 0,Y 608.418,Z 297.442,A -85,B 0,C 180,E1 -425.428,E2 -425.428} C_VEL
LIN {X 0,Y 608.477,Z 306.107,A -85,B 0,C 180,E1 -427.953,E2 -427.953} C_VEL
LIN {X 0,Y 608.432,Z 316.01,A -85,B 0,C 180,E1 -430.78,E2 -430.78} C_VEL
LIN {X 0,Y 608.433,Z 325.408,A -85,B 0,C 180,E1 -433.421,E2 -433.421} C_VEL
LIN {X 0,Y 608.669,Z 329.645,A -85,B 0,C 180,E1 -433.487,E2 -433.487} C_VEL
LIN {X 0,Y 608.678,Z 344.777,A -85,B 0,C 180,E1 -433.748,E2 -433.748} C_VEL
LIN {X 0,Y 608.642,Z 359.316,A -85,B 0,C 180,E1 -434.127,E2 -434.127} C_VEL
LIN {X 0,Y 608.586,Z 373.804,A -85,B 0,C 180,E1 -434.64,E2 -434.64} C_VEL
LIN {X 0,Y 608.573,Z 387.869,A -85,B 0,C 180,E1 -435.282,E2 -435.282} C_VEL
LIN {X 0,Y 608.562,Z 401.454,A -85,B 0,C 180,E1 -436.05,E2 -436.05} C_VEL
LIN {X 0,Y 608.547,Z 413.86,A -85,B 0,C 180,E1 -436.901,E2 -436.901} C_VEL
LIN {X 0,Y 608.522,Z 425.28,A -85,B 0,C 180,E1 -437.833,E2 -437.833} C_VEL
LIN {X 0,Y 608.492,Z 436.655,A -85,B 0,C 180,E1 -438.937,E2 -438.937} C_VEL
LIN {X 0,Y 608.471,Z 447.374,A -85,B 0,C 180,E1 -440.191,E2 -440.191} C_VEL
LIN {X 0,Y 608.464,Z 455.657,A -85,B 0,C 180,E1 -441.365,E2 -441.365} C_VEL
LIN {X 0,Y 608.456,Z 463.428,A -85,B 0,C 180,E1 -442.701,E2 -442.701} C_VEL
LIN {X 0,Y 608.437,Z 469.61,A -85,B 0,C 180,E1 -444.033,E2 -444.033} C_VEL
LIN {X 0,Y 608.427,Z 474.384,A -85,B 0,C 180,E1 -445.363,E2 -445.363} C_VEL
LIN {X 0,Y 608.421,Z 477.886,A -85,B 0,C 180,E1 -446.689,E2 -446.689} C_VEL
LIN {X 0,Y 608.444,Z 480.192,A -85,B 0,C 180,E1 -448.015,E2 -448.015} C_VEL
LIN {X 0,Y 608.434,Z 481.351,A -85,B 0,C 180,E1 -449.339,E2 -449.339} C_VEL
LIN {X 0,Y 608.434,Z 481.35,A -85,B 0,C 180,E1 -450.662,E2 -450.662} C_VEL
LIN {X 0,Y 608.444,Z 480.191,A -85,B 0,C 180,E1 -451.986,E2 -451.986} C_VEL
LIN {X 0,Y 608.421,Z 477.884,A -85,B 0,C 180,E1 -453.311,E2 -453.311} C_VEL
LIN {X 0,Y 608.427,Z 474.381,A -85,B 0,C 180,E1 -454.638,E2 -454.638} C_VEL
LIN {X 0,Y 608.437,Z 469.606,A -85,B 0,C 180,E1 -455.968,E2 -455.968} C_VEL
LIN {X 0,Y 608.456,Z 463.423,A -85,B 0,C 180,E1 -457.3,E2 -457.3} C_VEL
LIN {X 0,Y 608.464,Z 455.651,A -85,B 0,C 180,E1 -458.636,E2 -458.636} C_VEL
LIN {X 0,Y 608.471,Z 447.367,A -85,B 0,C 180,E1 -459.81,E2 -459.81} C_VEL
LIN {X 0,Y 608.492,Z 436.651,A -85,B 0,C 180,E1 -461.063,E2 -461.063} C_VEL
LIN {X 0,Y 608.522,Z 425.269,A -85,B 0,C 180,E1 -462.168,E2 -462.168} C_VEL
LIN {X 0,Y 608.547,Z 413.847,A -85,B 0,C 180,E1 -463.1,E2 -463.1} C_VEL
LIN {X 0,Y 608.564,Z 401.439,A -85,B 0,C 180,E1 -463.95,E2 -463.95} C_VEL
LIN {X 0,Y 608.573,Z 387.849,A -85,B 0,C 180,E1 -464.718,E2 -464.718} C_VEL
LIN {X 0,Y 608.586,Z 373.779,A -85,B 0,C 180,E1 -465.36,E2 -465.36} C_VEL
LIN {X 0,Y 608.659,Z 358.549,A -85,B 0,C 180,E1 -465.895,E2 -465.895} C_VEL
LIN {X 0,Y 608.689,Z 343.224,A -85,B 0,C 180,E1 -466.286,E2 -466.286} C_VEL
LIN {X 0,Y 608.694,Z 327.951,A -85,B 0,C 180,E1 -466.535,E2 -466.535} C_VEL
LIN {X 0,Y 608.441,Z 325.392,A -85,B 0,C 180,E1 -466.584,E2 -466.584} C_VEL
LIN {X 0,Y 608.433,Z 316.006,A -85,B 0,C 180,E1 -469.221,E2 -469.221} C_VEL
LIN {X 0,Y 608.477,Z 306.104,A -85,B 0,C 180,E1 -472.048,E2 -472.048} C_VEL
LIN {X 0,Y 608.419,Z 297.439,A -85,B 0,C 180,E1 -474.573,E2 -474.573} C_VEL
LIN {X 0,Y 608.418,Z 290.012,A -85,B 0,C 180,E1 -476.776,E2 -476.776} C_VEL
LIN {X 0,Y 608.503,Z 281.348,A -85,B 0,C 180,E1 -479.398,E2 -479.398} C_VEL
LIN {X 0,Y 608.446,Z 272.683,A -85,B 0,C 180,E1 -482.096,E2 -482.096} C_VEL
LIN {X 0,Y 608.454,Z 265.256,A -85,B 0,C 180,E1 -484.471,E2 -484.471} C_VEL
LIN {X 0,Y 608.515,Z 257.829,A -85,B 0,C 180,E1 -486.911,E2 -486.911} C_VEL
LIN {X 0,Y 608.529,Z 249.165,A -85,B 0,C 180,E1 -489.865,E2 -489.865} C_VEL
LIN {X 0,Y 608.47,Z 244.319,A -85,B 0,C 180,E1 -491.6,E2 -491.6} C_VEL
LIN {X 0,Y 608.464,Z 244.321,A -85,B 0,C 180,E1 -494.264,E2 -494.264} C_VEL
LIN {X 0,Y 608.449,Z 244.321,A -85,B 0,C 180,E1 -497.04,E2 -497.04} C_VEL
LIN {X 0,Y 608.457,Z 244.32,A -85,B 0,C 180,E1 -499.697,E2 -499.697} C_VEL
LIN {X 0,Y 608.465,Z 244.319,A -85,B 0,C 180,E1 -502.253,E2 -502.253} C_VEL
LIN {X 0,Y 608.458,Z 244.32,A -85,B 0,C 180,E1 -505.094,E2 -505.094} C_VEL
LIN {X 0,Y 608.468,Z 244.32,A -85,B 0,C 180,E1 -507.905,E2 -507.905} C_VEL
LIN {X 0,Y 608.46,Z 244.32,A -85,B 0,C 180,E1 -510.22,E2 -510.22} C_VEL
LIN {X 0,Y 608.485,Z 244.317,A -85,B 0,C 180,E1 -512.792,E2 -512.792} C_VEL
LIN {X 0,Y 608.454,Z 244.321,A -85,B 0,C 180,E1 -515.429,E2 -515.429} C_VEL
LIN {X 0,Y 608.468,Z 244.321,A -85,B 0,C 180,E1 -518.308,E2 -518.308} C_VEL
LIN {X 0,Y 608.477,Z 244.319,A -85,B 0,C 180,E1 -521.283,E2 -521.283} C_VEL
LIN {X 0,Y 608.455,Z 244.32,A -85,B 0,C 180,E1 -523.906,E2 -523.906} C_VEL
LIN {X 0,Y 608.467,Z 244.321,A -85,B 0,C 180,E1 -526.643,E2 -526.643} C_VEL
LIN {X 0,Y 608.458,Z 244.32,A -85,B 0,C 180,E1 -529.349,E2 -529.349} C_VEL
LIN {X 0,Y 608.477,Z 244.318,A -85,B 0,C 180,E1 -532.032,E2 -532.032} C_VEL
LIN {X 0,Y 608.475,Z 244.318,A -85,B 0,C 180,E1 -534.698,E2 -534.698} C_VEL
LIN {X 0,Y 608.471,Z 244.318,A -85,B 0,C 180,E1 -537.351,E2 -537.351} C_VEL
LIN {X 0,Y 608.476,Z 244.319,A -85,B 0,C 180,E1 -539.999,E2 -539.999} C_VEL
LIN {X 0,Y 608.481,Z 244.317,A -85,B 0,C 180,E1 -542.647,E2 -542.647} C_VEL
LIN {X 0,Y 608.466,Z 244.321,A -85,B 0,C 180,E1 -545.301,E2 -545.301} C_VEL
LIN {X 0,Y 608.477,Z 244.317,A -85,B 0,C 180,E1 -547.966,E2 -547.966} C_VEL
LIN {X 0,Y 608.453,Z 244.32,A -85,B 0,C 180,E1 -549.458,E2 -549.458} C_VEL
LIN {X 0,Y 607.78,Z 244.405,A -85,B 0,C 180,E1 -550.011,E2 -550.011} C_VEL
LIN {X 0,Y 604.931,Z 244.76,A -85,B 0,C 180,E1 -550.908,E2 -550.908} C_VEL
LIN {X 0,Y 602.53,Z 245.06,A -85,B 0,C 180,E1 -551.629,E2 -551.629} C_VEL
LIN {X 0,Y 601.499,Z 245.187,A -85,B 0,C 180,E1 -552.186,E2 -552.186} C_VEL
LIN {X 0,Y 601.414,Z 245.197,A -85,B 0,C 180,E1 -552.374,E2 -552.374} C_VEL
LIN {X 0,Y 601.429,Z 245.197,A -85,B 0,C 180,E1 -554.896,E2 -554.896} C_VEL
LIN {X 0,Y 601.431,Z 245.197,A -85,B 0,C 180,E1 -556.985,E2 -556.985} C_VEL
LIN {X 0,Y 601.404,Z 245.199,A -85,B 0,C 180,E1 -559.808,E2 -559.808} C_VEL
LIN {X 0,Y 601.412,Z 245.197,A -85,B 0,C 180,E1 -562.682,E2 -562.682} C_VEL
LIN {X 0,Y 601.402,Z 245.199,A -85,B 0,C 180,E1 -564.877,E2 -564.877} C_VEL
LIN {X 0,Y 601.424,Z 245.196,A -85,B 0,C 180,E1 -567.866,E2 -567.866} C_VEL
LIN {X 0,Y 601.427,Z 245.196,A -85,B 0,C 180,E1 -570.163,E2 -570.163} C_VEL
LIN {X 0,Y 601.421,Z 245.198,A -85,B 0,C 180,E1 -572.715,E2 -572.715} C_VEL
LIN {X 0,Y 601.413,Z 245.197,A -85,B 0,C 180,E1 -575.114,E2 -575.114} C_VEL
LIN {X 0,Y 601.431,Z 245.195,A -85,B 0,C 180,E1 -577.418,E2 -577.418} C_VEL
LIN {X 0,Y 601.408,Z 245.2,A -85,B 0,C 180,E1 -579.994,E2 -579.994} C_VEL
LIN {X 0,Y 601.408,Z 245.198,A -85,B 0,C 180,E1 -582.669,E2 -582.669} C_VEL
LIN {X 0,Y 601.42,Z 245.197,A -85,B 0,C 180,E1 -585.481,E2 -585.481} C_VEL
LIN {X 0,Y 601.42,Z 245.198,A -85,B 0,C 180,E1 -588.405,E2 -588.405} C_VEL
LIN {X 0,Y 601.428,Z 245.195,A -85,B 0,C 180,E1 -590.874,E2 -590.874} C_VEL
LIN {X 0,Y 601.437,Z 245.195,A -85,B 0,C 180,E1 -593.733,E2 -593.733} C_VEL
LIN {X 0,Y 601.425,Z 245.198,A -85,B 0,C 180,E1 -596.686,E2 -596.686} C_VEL
LIN {X 0,Y 601.428,Z 245.196,A -85,B 0,C 180,E1 -599.058,E2 -599.058} C_VEL
LIN {X 0,Y 601.435,Z 245.194,A -85,B 0,C 180,E1 -601.373,E2 -601.373} C_VEL
LIN {X 0,Y 601.405,Z 245.199,A -85,B 0,C 180,E1 -603.636,E2 -603.636} C_VEL
LIN {X 0,Y 601.419,Z 245.196,A -85,B 0,C 180,E1 -606.589,E2 -606.589} C_VEL
LIN {X 0,Y 601.432,Z 245.196,A -85,B 0,C 180,E1 -609.478,E2 -609.478} C_VEL
LIN {X 0,Y 601.391,Z 245.203,A -85,B 0,C 180,E1 -612.311,E2 -612.311} C_VEL
LIN {X 0,Y 601.41,Z 245.2,A -85,B 0,C 180,E1 -614.408,E2 -614.408} C_VEL
LIN {X 0,Y 601.422,Z 245.196,A -85,B 0,C 180,E1 -617.171,E2 -617.171} C_VEL
LIN {X 0,Y 601.428,Z 245.196,A -85,B 0,C 180,E1 -619.904,E2 -619.904} C_VEL
LIN {X 0,Y 601.448,Z 245.194,A -85,B 0,C 180,E1 -622.615,E2 -622.615} C_VEL
LIN {X 0,Y 601.428,Z 245.196,A -85,B 0,C 180,E1 -624.635,E2 -624.635} C_VEL
LIN {X 0,Y 601.373,Z 245.382,A -85,B 0,C 180,E1 -625.307,E2 -625.307} C_VEL
LIN {X 0,Y 601.408,Z 248.19,A -85,B 0,C 180,E1 -627.99,E2 -627.99} C_VEL
LIN {X 0,Y 601.363,Z 250.956,A -85,B 0,C 180,E1 -630.669,E2 -630.669} C_VEL
LIN {X 0,Y 601.33,Z 253.773,A -85,B 0,C 180,E1 -633.35,E2 -633.35} C_VEL
LIN {X 0,Y 601.293,Z 256.881,A -85,B 0,C 180,E1 -636.038,E2 -636.038} C_VEL
LIN {X 0,Y 601.305,Z 260.076,A -85,B 0,C 180,E1 -638.739,E2 -638.739} C_VEL
LIN {X 0,Y 601.291,Z 263.366,A -85,B 0,C 180,E1 -641.46,E2 -641.46} C_VEL
LIN {X 0,Y 601.283,Z 266.752,A -85,B 0,C 180,E1 -644.208,E2 -644.208} C_VEL
LIN {X 0,Y 601.296,Z 269.388,A -85,B 0,C 180,E1 -646.318,E2 -646.318} C_VEL
LIN {X 0,Y 601.892,Z 273.606,A -85,B 0,C 180,E1 -646.398,E2 -646.398} C_VEL
LIN {X 0,Y 601.829,Z 288.933,A -85,B 0,C 180,E1 -646.702,E2 -646.702} C_VEL
LIN {X 0,Y 601.736,Z 303.002,A -85,B 0,C 180,E1 -647.108,E2 -647.108} C_VEL
LIN {X 0,Y 601.654,Z 317.87,A -85,B 0,C 180,E1 -647.68,E2 -647.68} C_VEL
LIN {X 0,Y 601.656,Z 332.13,A -85,B 0,C 180,E1 -648.384,E2 -648.384} C_VEL
LIN {X 0,Y 601.612,Z 345.262,A -85,B 0,C 180,E1 -649.181,E2 -649.181} C_VEL
LIN {X 0,Y 601.542,Z 357.455,A -85,B 0,C 180,E1 -650.071,E2 -650.071} C_VEL
LIN {X 0,Y 601.504,Z 369.176,A -85,B 0,C 180,E1 -651.095,E2 -651.095} C_VEL
LIN {X 0,Y 601.444,Z 379.236,A -85,B 0,C 180,E1 -652.137,E2 -652.137} C_VEL
LIN {X 0,Y 601.434,Z 388.158,A -85,B 0,C 180,E1 -653.227,E2 -653.227} C_VEL
LIN {X 0,Y 601.396,Z 395.525,A -85,B 0,C 180,E1 -654.287,E2 -654.287} C_VEL
LIN {X 0,Y 601.365,Z 403.216,A -85,B 0,C 180,E1 -655.62,E2 -655.62} C_VEL
LIN {X 0,Y 601.352,Z 408.478,A -85,B 0,C 180,E1 -656.74,E2 -656.74} C_VEL
LIN {X 0,Y 601.349,Z 412.855,A -85,B 0,C 180,E1 -657.87,E2 -657.87} C_VEL
LIN {X 0,Y 601.338,Z 415.629,A -85,B 0,C 180,E1 -658.775,E2 -658.775} C_VEL
LIN {X 0,Y 601.328,Z 418.861,A -85,B 0,C 180,E1 -660.169,E2 -660.169} C_VEL
LIN {X 0,Y 601.318,Z 420.93,A -85,B 0,C 180,E1 -661.731,E2 -661.731} C_VEL
LIN {X 0,Y 601.323,Z 421.427,A -85,B 0,C 180,E1 -662.703,E2 -662.703} C_VEL
LIN {X 0,Y 601.316,Z 421.093,A -85,B 0,C 180,E1 -664.125,E2 -664.125} C_VEL
LIN {X 0,Y 601.316,Z 420.135,A -85,B 0,C 180,E1 -665.103,E2 -665.103} C_VEL
LIN {X 0,Y 601.33,Z 417.475,A -85,B 0,C 180,E1 -666.587,E2 -666.587} C_VEL
LIN {X 0,Y 601.339,Z 414.035,A -85,B 0,C 180,E1 -667.848,E2 -667.848} C_VEL
LIN {X 0,Y 601.344,Z 409.404,A -85,B 0,C 180,E1 -669.131,E2 -669.131} C_VEL
LIN {X 0,Y 601.368,Z 404.186,A -85,B 0,C 180,E1 -670.282,E2 -670.282} C_VEL
LIN {X 0,Y 601.383,Z 396.859,A -85,B 0,C 180,E1 -671.591,E2 -671.591} C_VEL
LIN {X 0,Y 601.42,Z 387.914,A -85,B 0,C 180,E1 -672.897,E2 -672.897} C_VEL
LIN {X 0,Y 601.475,Z 378.423,A -85,B 0,C 180,E1 -674.045,E2 -674.045} C_VEL
LIN {X 0,Y 601.483,Z 367.872,A -85,B 0,C 180,E1 -675.121,E2 -675.121} C_VEL
LIN {X 0,Y 601.543,Z 356.712,A -85,B 0,C 180,E1 -676.079,E2 -676.079} C_VEL
LIN {X 0,Y 601.59,Z 343.856,A -85,B 0,C 180,E1 -677.005,E2 -677.005} C_VEL
LIN {X 0,Y 601.67,Z 330.295,A -85,B 0,C 180,E1 -677.807,E2 -677.807} C_VEL
LIN {X 0,Y 601.718,Z 316.125,A -85,B 0,C 180,E1 -678.485,E2 -678.485} C_VEL
LIN {X 0,Y 601.759,Z 302.769,A -85,B 0,C 180,E1 -678.989,E2 -678.989} C_VEL
LIN {X 0,Y 601.843,Z 287.524,A -85,B 0,C 180,E1 -679.421,E2 -679.421} C_VEL
LIN {X 0,Y 601.766,Z 271.639,A -85,B 0,C 180,E1 -679.724,E2 -679.724} C_VEL
LIN {X 0,Y 601.337,Z 269.386,A -85,B 0,C 180,E1 -679.773,E2 -679.773} C_VEL
LIN {X 0,Y 601.318,Z 265.82,A -85,B 0,C 180,E1 -682.632,E2 -682.632} C_VEL
LIN {X 0,Y 601.351,Z 262.833,A -85,B 0,C 180,E1 -685.065,E2 -685.065} C_VEL
LIN {X 0,Y 601.331,Z 259.921,A -85,B 0,C 180,E1 -687.479,E2 -687.479} C_VEL
LIN {X 0,Y 601.351,Z 257.099,A -85,B 0,C 180,E1 -689.863,E2 -689.863} C_VEL
LIN {X 0,Y 601.341,Z 253.608,A -85,B 0,C 180,E1 -692.885,E2 -692.885} C_VEL
LIN {X 0,Y 601.387,Z 250.78,A -85,B 0,C 180,E1 -695.716,E2 -695.716} C_VEL
LIN {X 0,Y 601.371,Z 247.743,A -85,B 0,C 180,E1 -698.76,E2 -698.76} C_VEL
LIN {X 0,Y 601.392,Z 245.203,A -85,B 0,C 180,E1 -701.186,E2 -701.186} C_VEL
LIN {X 0,Y 601.44,Z 245.195,A -85,B 0,C 180,E1 -703.714,E2 -703.714} C_VEL
LIN {X 0,Y 601.416,Z 245.198,A -85,B 0,C 180,E1 -706.485,E2 -706.485} C_VEL
LIN {X 0,Y 601.417,Z 245.197,A -85,B 0,C 180,E1 -709.225,E2 -709.225} C_VEL
LIN {X 0,Y 601.438,Z 245.197,A -85,B 0,C 180,E1 -711.94,E2 -711.94} C_VEL
LIN {X 0,Y 601.423,Z 245.196,A -85,B 0,C 180,E1 -714.637,E2 -714.637} C_VEL
LIN {X 0,Y 601.448,Z 245.195,A -85,B 0,C 180,E1 -717.322,E2 -717.322} C_VEL
LIN {X 0,Y 601.442,Z 245.194,A -85,B 0,C 180,E1 -720.001,E2 -720.001} C_VEL
LIN {X 0,Y 601.445,Z 245.194,A -85,B 0,C 180,E1 -722.68,E2 -722.68} C_VEL
LIN {X 0,Y 601.43,Z 245.196,A -85,B 0,C 180,E1 -725.365,E2 -725.365} C_VEL
LIN {X 0,Y 601.438,Z 245.195,A -85,B 0,C 180,E1 -728.061,E2 -728.061} C_VEL
LIN {X 0,Y 601.424,Z 245.198,A -85,B 0,C 180,E1 -731.015,E2 -731.015} C_VEL
LIN {X 0,Y 601.423,Z 245.196,A -85,B 0,C 180,E1 -733.516,E2 -733.516} C_VEL
LIN {X 0,Y 601.436,Z 245.196,A -85,B 0,C 180,E1 -736.288,E2 -736.288} C_VEL
LIN {X 0,Y 601.416,Z 245.197,A -85,B 0,C 180,E1 -739.099,E2 -739.099} C_VEL
LIN {X 0,Y 601.41,Z 245.198,A -85,B 0,C 180,E1 -741.24,E2 -741.24} C_VEL
LIN {X 0,Y 601.448,Z 245.193,A -85,B 0,C 180,E1 -744.141,E2 -744.141} C_VEL
LIN {X 0,Y 601.456,Z 245.192,A -85,B 0,C 180,E1 -747.111,E2 -747.111} C_VEL
LIN {X 0,Y 601.42,Z 245.196,A -85,B 0,C 180,E1 -749.393,E2 -749.393} C_VEL
LIN {X 0,Y 601.399,Z 245.2,A -85,B 0,C 180,E1 -751.727,E2 -751.727} C_VEL
LIN {X 0,Y 601.429,Z 245.198,A -85,B 0,C 180,E1 -754.119,E2 -754.119} C_VEL
LIN {X 0,Y 601.436,Z 245.197,A -85,B 0,C 180,E1 -757.383,E2 -757.383} C_VEL
LIN {X 0,Y 601.408,Z 245.198,A -85,B 0,C 180,E1 -759.996,E2 -759.996} C_VEL
LIN {X 0,Y 601.409,Z 245.2,A -85,B 0,C 180,E1 -762.671,E2 -762.671} C_VEL
LIN {X 0,Y 601.424,Z 245.197,A -85,B 0,C 180,E1 -765.483,E2 -765.483} C_VEL
LIN {X 0,Y 601.459,Z 245.294,A -85,B 0,C 180,E1 -768.183,E2 -768.183} C_VEL
LIN {X 0,Y 601.582,Z 248.682,A -85,B 0,C 180,E1 -769.408,E2 -769.408} C_VEL
LIN {X 0,Y 601.551,Z 255.357,A -85,B 0,C 180,E1 -771.743,E2 -771.743} C_VEL
LIN {X 0,Y 601.538,Z 262.784,A -85,B 0,C 180,E1 -774.256,E2 -774.256} C_VEL
LIN {X 0,Y 601.524,Z 270.211,A -85,B 0,C 180,E1 -776.693,E2 -776.693} C_VEL
LIN {X 0,Y 601.491,Z 277.638,A -85,B 0,C 180,E1 -779.063,E2 -779.063} C_VEL
LIN {X 0,Y 601.447,Z 286.302,A -85,B 0,C 180,E1 -781.755,E2 -781.755} C_VEL
LIN {X 0,Y 601.43,Z 296.205,A -85,B 0,C 180,E1 -784.754,E2 -784.754} C_VEL
LIN {X 0,Y 601.4,Z 305.146,A -85,B 0,C 180,E1 -787.398,E2 -787.398} C_VEL
LIN {X 0,Y 601.412,Z 314.772,A -85,B 0,C 180,E1 -790.191,E2 -790.191} C_VEL
LIN {X 0,Y 601.376,Z 323.436,A -85,B 0,C 180,E1 -792.663,E2 -792.663} C_VEL
LIN {X 0,Y 601.368,Z 325.398,A -85,B 0,C 180,E1 -793.217,E2 -793.217} C_VEL
LIN {X 0,Y 601.878,Z 329.927,A -85,B 0,C 180,E1 -793.299,E2 -793.299} C_VEL
LIN {X 0,Y 601.866,Z 344.876,A -85,B 0,C 180,E1 -793.561,E2 -793.561} C_VEL
LIN {X 0,Y 601.805,Z 359.316,A -85,B 0,C 180,E1 -793.942,E2 -793.942} C_VEL
LIN {X 0,Y 601.703,Z 373.805,A -85,B 0,C 180,E1 -794.46,E2 -794.46} C_VEL
LIN {X 0,Y 601.661,Z 387.87,A -85,B 0,C 180,E1 -795.109,E2 -795.109} C_VEL
LIN {X 0,Y 601.613,Z 401.592,A -85,B 0,C 180,E1 -795.894,E2 -795.894} C_VEL
LIN {X 0,Y 601.57,Z 415.02,A -85,B 0,C 180,E1 -796.832,E2 -796.832} C_VEL
LIN {X 0,Y 601.513,Z 427.198,A -85,B 0,C 180,E1 -797.86,E2 -797.86} C_VEL
LIN {X 0,Y 601.437,Z 438.277,A -85,B 0,C 180,E1 -798.983,E2 -798.983} C_VEL
LIN {X 0,Y 601.428,Z 447.374,A -85,B 0,C 180,E1 -800.075,E2 -800.075} C_VEL
LIN {X 0,Y 601.386,Z 455.657,A -85,B 0,C 180,E1 -801.262,E2 -801.262} C_VEL
LIN {X 0,Y 601.365,Z 463.429,A -85,B 0,C 180,E1 -802.614,E2 -802.614} C_VEL
LIN {X 0,Y 601.357,Z 469.609,A -85,B 0,C 180,E1 -803.963,E2 -803.963} C_VEL
LIN {X 0,Y 601.33,Z 474.384,A -85,B 0,C 180,E1 -805.308,E2 -805.308} C_VEL
LIN {X 0,Y 601.337,Z 477.887,A -85,B 0,C 180,E1 -806.65,E2 -806.65} C_VEL
LIN {X 0,Y 601.343,Z 480.192,A -85,B 0,C 180,E1 -807.991,E2 -807.991} C_VEL
LIN {X 0,Y 601.335,Z 481.35,A -85,B 0,C 180,E1 -809.331,E2 -809.331} C_VEL
LIN {X 0,Y 601.335,Z 481.35,A -85,B 0,C 180,E1 -810.67,E2 -810.67} C_VEL
LIN {X 0,Y 601.343,Z 480.191,A -85,B 0,C 180,E1 -812.01,E2 -812.01} C_VEL
LIN {X 0,Y 601.337,Z 477.885,A -85,B 0,C 180,E1 -813.351,E2 -813.351} C_VEL
LIN {X 0,Y 601.33,Z 474.382,A -85,B 0,C 180,E1 -814.693,E2 -814.693} C_VEL
LIN {X 0,Y 601.357,Z 469.606,A -85,B 0,C 180,E1 -816.038,E2 -816.038} C_VEL
LIN {X 0,Y 601.365,Z 463.423,A -85,B 0,C 180,E1 -817.386,E2 -817.386} C_VEL
LIN {X 0,Y 601.386,Z 455.651,A -85,B 0,C 180,E1 -818.739,E2 -818.739} C_VEL
LIN {X 0,Y 601.428,Z 447.367,A -85,B 0,C 180,E1 -819.926,E2 -819.926} C_VEL
LIN {X 0,Y 601.461,Z 436.931,A -85,B 0,C 180,E1 -821.165,E2 -821.165} C_VEL
LIN {X 0,Y 601.514,Z 427.188,A -85,B 0,C 180,E1 -822.141,E2 -822.141} C_VEL
LIN {X 0,Y 601.57,Z 415.008,A -85,B 0,C 180,E1 -823.169,E2 -823.169} C_VEL
LIN {X 0,Y 601.608,Z 403.073,A -85,B 0,C 180,E1 -824.012,E2 -824.012} C_VEL
LIN {X 0,Y 601.674,Z 389.521,A -85,B 0,C 180,E1 -824.805,E2 -824.805} C_VEL
LIN {X 0,Y 601.716,Z 374.835,A -85,B 0,C 180,E1 -825.497,E2 -825.497} C_VEL
LIN {X 0,Y 601.792,Z 360.605,A -85,B 0,C 180,E1 -826.016,E2 -826.016} C_VEL
LIN {X 0,Y 601.838,Z 345.718,A -85,B 0,C 180,E1 -826.42,E2 -826.42} C_VEL
LIN {X 0,Y 601.86,Z 330.419,A -85,B 0,C 180,E1 -826.694,E2 -826.694} C_VEL
LIN {X 0,Y 601.558,Z 326.608,A -85,B 0,C 180,E1 -826.754,E2 -826.754} C_VEL
LIN {X 0,Y 601.371,Z 325.391,A -85,B 0,C 180,E1 -826.784,E2 -826.784} C_VEL
LIN {X 0,Y 601.413,Z 316.006,A -85,B 0,C 180,E1 -829.454,E2 -829.454} C_VEL
LIN {X 0,Y 601.426,Z 306.242,A -85,B 0,C 180,E1 -832.28,E2 -832.28} C_VEL
LIN {X 0,Y 601.394,Z 297.439,A -85,B 0,C 180,E1 -834.879,E2 -834.879} C_VEL
LIN {X 0,Y 601.444,Z 289.172,A -85,B 0,C 180,E1 -837.367,E2 -837.367} C_VEL
LIN {X 0,Y 601.449,Z 280.11,A -85,B 0,C 180,E1 -840.163,E2 -840.163} C_VEL
LIN {X 0,Y 601.449,Z 272.683,A -85,B 0,C 180,E1 -842.515,E2 -842.515} C_VEL
LIN {X 0,Y 601.544,Z 264.626,A -85,B 0,C 180,E1 -845.132,E2 -845.132} C_VEL
LIN {X 0,Y 601.579,Z 256.592,A -85,B 0,C 180,E1 -847.832,E2 -847.832} C_VEL
LIN {X 0,Y 601.585,Z 248.681,A -85,B 0,C 180,E1 -850.592,E2 -850.592} C_VEL
LIN {X 0,Y 601.424,Z 245.197,A -85,B 0,C 180,E1 -851.878,E2 -851.878} C_VEL
LIN {X 0,Y 601.429,Z 245.196,A -85,B 0,C 180,E1 -854.535,E2 -854.535} C_VEL
LIN {X 0,Y 601.411,Z 245.2,A -85,B 0,C 180,E1 -857.41,E2 -857.41} C_VEL
LIN {X 0,Y 601.406,Z 245.198,A -85,B 0,C 180,E1 -860.004,E2 -860.004} C_VEL
LIN {X 0,Y 601.441,Z 245.196,A -85,B 0,C 180,E1 -862.618,E2 -862.618} C_VEL
LIN {X 0,Y 601.418,Z 245.197,A -85,B 0,C 180,E1 -865.068,E2 -865.068} C_VEL
LIN {X 0,Y 601.434,Z 245.195,A -85,B 0,C 180,E1 -867.484,E2 -867.484} C_VEL
LIN {X 0,Y 601.433,Z 245.197,A -85,B 0,C 180,E1 -869.851,E2 -869.851} C_VEL
LIN {X 0,Y 601.456,Z 245.194,A -85,B 0,C 180,E1 -872.889,E2 -872.889} C_VEL
LIN {X 0,Y 601.453,Z 245.193,A -85,B 0,C 180,E1 -875.859,E2 -875.859} C_VEL
LIN {X 0,Y 601.411,Z 245.197,A -85,B 0,C 180,E1 -878.76,E2 -878.76} C_VEL
LIN {X 0,Y 601.421,Z 245.197,A -85,B 0,C 180,E1 -881.608,E2 -881.608} C_VEL
LIN {X 0,Y 601.415,Z 245.199,A -85,B 0,C 180,E1 -884.408,E2 -884.408} C_VEL
LIN {X 0,Y 601.422,Z 245.196,A -85,B 0,C 180,E1 -887.171,E2 -887.171} C_VEL
LIN {X 0,Y 601.429,Z 245.197,A -85,B 0,C 180,E1 -889.904,E2 -889.904} C_VEL
LIN {X 0,Y 601.447,Z 245.194,A -85,B 0,C 180,E1 -892.614,E2 -892.614} C_VEL
LIN {X 0,Y 601.416,Z 245.197,A -85,B 0,C 180,E1 -895.307,E2 -895.307} C_VEL
LIN {X 0,Y 601.433,Z 245.197,A -85,B 0,C 180,E1 -897.99,E2 -897.99} C_VEL
LIN {X 0,Y 601.454,Z 245.192,A -85,B 0,C 180,E1 -900.669,E2 -900.669} C_VEL
LIN {X 0,Y 601.43,Z 245.198,A -85,B 0,C 180,E1 -903.349,E2 -903.349} C_VEL
LIN {X 0,Y 601.408,Z 245.198,A -85,B 0,C 180,E1 -906.036,E2 -906.036} C_VEL
LIN {X 0,Y 601.419,Z 245.198,A -85,B 0,C 180,E1 -908.737,E2 -908.737} C_VEL
LIN {X 0,Y 601.417,Z 245.198,A -85,B 0,C 180,E1 -911.458,E2 -911.458} C_VEL
LIN {X 0,Y 601.414,Z 245.197,A -85,B 0,C 180,E1 -912.374,E2 -912.374} C_VEL
LIN {X 0,Y 600.747,Z 245.282,A -85,B 0,C 180,E1 -912.933,E2 -912.933} C_VEL
LIN {X 0,Y 597.895,Z 245.638,A -85,B 0,C 180,E1 -913.841,E2 -913.841} C_VEL
LIN {X 0,Y 595.484,Z 245.937,A -85,B 0,C 180,E1 -914.571,E2 -914.571} C_VEL
LIN {X 0,Y 594.446,Z 246.066,A -85,B 0,C 180,E1 -915.135,E2 -915.135} C_VEL
LIN {X 0,Y 594.36,Z 246.075,A -85,B 0,C 180,E1 -915.326,E2 -915.326} C_VEL
LIN {X 0,Y 594.38,Z 246.076,A -85,B 0,C 180,E1 -917.903,E2 -917.903} C_VEL
LIN {X 0,Y 594.374,Z 246.075,A -85,B 0,C 180,E1 -920.914,E2 -920.914} C_VEL
LIN {X 0,Y 594.391,Z 246.072,A -85,B 0,C 180,E1 -923.703,E2 -923.703} C_VEL
LIN {X 0,Y 594.382,Z 246.073,A -85,B 0,C 180,E1 -926.698,E2 -926.698} C_VEL
LIN {X 0,Y 594.382,Z 246.073,A -85,B 0,C 180,E1 -928.997,E2 -928.997} C_VEL
LIN {X 0,Y 594.384,Z 246.075,A -85,B 0,C 180,E1 -931.643,E2 -931.643} C_VEL
LIN {X 0,Y 594.395,Z 246.073,A -85,B 0,C 180,E1 -934.578,E2 -934.578} C_VEL
LIN {X 0,Y 594.382,Z 246.073,A -85,B 0,C 180,E1 -937.085,E2 -937.085} C_VEL
LIN {X 0,Y 594.373,Z 246.076,A -85,B 0,C 180,E1 -939.773,E2 -939.773} C_VEL
LIN {X 0,Y 594.366,Z 246.075,A -85,B 0,C 180,E1 -942.374,E2 -942.374} C_VEL
LIN {X 0,Y 594.358,Z 246.079,A -85,B 0,C 180,E1 -945.19,E2 -945.19} C_VEL
LIN {X 0,Y 594.383,Z 246.073,A -85,B 0,C 180,E1 -947.625,E2 -947.625} C_VEL
LIN {X 0,Y 594.388,Z 246.075,A -85,B 0,C 180,E1 -950.32,E2 -950.32} C_VEL
LIN {X 0,Y 594.379,Z 246.073,A -85,B 0,C 180,E1 -952.912,E2 -952.912} C_VEL
LIN {X 0,Y 594.376,Z 246.075,A -85,B 0,C 180,E1 -955.86,E2 -955.86} C_VEL
LIN {X 0,Y 594.386,Z 246.075,A -85,B 0,C 180,E1 -958.65,E2 -958.65} C_VEL
LIN {X 0,Y 594.38,Z 246.074,A -85,B 0,C 180,E1 -961.04,E2 -961.04} C_VEL
LIN {X 0,Y 594.381,Z 246.076,A -85,B 0,C 180,E1 -963.975,E2 -963.975} C_VEL
LIN {X 0,Y 594.39,Z 246.073,A -85,B 0,C 180,E1 -966.296,E2 -966.296} C_VEL
LIN {X 0,Y 594.403,Z 246.073,A -85,B 0,C 180,E1 -969.224,E2 -969.224} C_VEL
LIN {X 0,Y 594.373,Z 246.075,A -85,B 0,C 180,E1 -972.095,E2 -972.095} C_VEL
LIN {X 0,Y 594.363,Z 246.077,A -85,B 0,C 180,E1 -974.219,E2 -974.219} C_VEL
LIN {X 0,Y 594.368,Z 246.075,A -85,B 0,C 180,E1 -977.017,E2 -977.017} C_VEL
LIN {X 0,Y 594.39,Z 246.073,A -85,B 0,C 180,E1 -979.784,E2 -979.784} C_VEL
LIN {X 0,Y 594.411,Z 246.07,A -85,B 0,C 180,E1 -982.527,E2 -982.527} C_VEL
LIN {X 0,Y 594.315,Z 246.084,A -85,B 0,C 180,E1 -985.251,E2 -985.251} C_VEL
LIN {X 0,Y 594.354,Z 248.765,A -85,B 0,C 180,E1 -987.967,E2 -987.967} C_VEL
LIN {X 0,Y 594.311,Z 251.551,A -85,B 0,C 180,E1 -990.677,E2 -990.677} C_VEL
LIN {X 0,Y 594.246,Z 254.346,A -85,B 0,C 180,E1 -993.39,E2 -993.39} C_VEL
LIN {X 0,Y 594.25,Z 256.579,A -85,B 0,C 180,E1 -995.429,E2 -995.429} C_VEL
LIN {X 0,Y 594.218,Z 259.757,A -85,B 0,C 180,E1 -998.159,E2 -998.159} C_VEL
LIN {X 0,Y 594.232,Z 263.14,A -85,B 0,C 180,E1 -1001.003,E2 -1001.003} C_VEL
LIN {X 0,Y 594.217,Z 266.92,A -85,B 0,C 180,E1 -1004.113,E2 -1004.113} C_VEL
LIN {X 0,Y 594.215,Z 269.412,A -85,B 0,C 180,E1 -1006.115,E2 -1006.115} C_VEL
LIN {X 0,Y 595.08,Z 273.55,A -85,B 0,C 180,E1 -1006.201,E2 -1006.201} C_VEL
LIN {X 0,Y 595.011,Z 288.94,A -85,B 0,C 180,E1 -1006.509,E2 -1006.509} C_VEL
LIN {X 0,Y 594.911,Z 302.083,A -85,B 0,C 180,E1 -1006.889,E2 -1006.889} C_VEL
LIN {X 0,Y 594.795,Z 316.712,A -85,B 0,C 180,E1 -1007.447,E2 -1007.447} C_VEL
LIN {X 0,Y 594.766,Z 329.608,A -85,B 0,C 180,E1 -1008.07,E2 -1008.07} C_VEL
LIN {X 0,Y 594.671,Z 343.571,A -85,B 0,C 180,E1 -1008.9,E2 -1008.9} C_VEL
LIN {X 0,Y 594.573,Z 355.736,A -85,B 0,C 180,E1 -1009.776,E2 -1009.776} C_VEL
LIN {X 0,Y 594.525,Z 367.305,A -85,B 0,C 180,E1 -1010.771,E2 -1010.771} C_VEL
LIN {X 0,Y 594.426,Z 378.01,A -85,B 0,C 180,E1 -1011.865,E2 -1011.865} C_VEL
LIN {X 0,Y 594.377,Z 387.101,A -85,B 0,C 180,E1 -1012.966,E2 -1012.966} C_VEL
LIN {X 0,Y 594.337,Z 395.92,A -85,B 0,C 180,E1 -1014.243,E2 -1014.243} C_VEL
LIN {X 0,Y 594.302,Z 403.425,A -85,B 0,C 180,E1 -1015.571,E2 -1015.571} C_VEL
LIN {X 0,Y 594.282,Z 408.642,A -85,B 0,C 180,E1 -1016.704,E2 -1016.704} C_VEL
LIN {X 0,Y 594.258,Z 412.986,A -85,B 0,C 180,E1 -1017.848,E2 -1017.848} C_VEL
LIN {X 0,Y 594.245,Z 416.365,A -85,B 0,C 180,E1 -1019.005,E2 -1019.005} C_VEL
LIN {X 0,Y 594.224,Z 419.137,A -85,B 0,C 180,E1 -1020.304,E2 -1020.304} C_VEL
LIN {X 0,Y 594.218,Z 420.863,A -85,B 0,C 180,E1 -1021.62,E2 -1021.62} C_VEL
LIN {X 0,Y 594.236,Z 421.486,A -85,B 0,C 180,E1 -1022.958,E2 -1022.958} C_VEL
LIN {X 0,Y 594.24,Z 421.106,A -85,B 0,C 180,E1 -1024.121,E2 -1024.121} C_VEL
LIN {X 0,Y 594.22,Z 419.737,A -85,B 0,C 180,E1 -1025.417,E2 -1025.417} C_VEL
LIN {X 0,Y 594.229,Z 417.824,A -85,B 0,C 180,E1 -1026.465,E2 -1026.465} C_VEL
LIN {X 0,Y 594.263,Z 413.899,A -85,B 0,C 180,E1 -1027.949,E2 -1027.949} C_VEL
LIN {X 0,Y 594.257,Z 409.21,A -85,B 0,C 180,E1 -1029.25,E2 -1029.25} C_VEL
LIN {X 0,Y 594.272,Z 403.137,A -85,B 0,C 180,E1 -1030.574,E2 -1030.574} C_VEL
LIN {X 0,Y 594.306,Z 395.955,A -85,B 0,C 180,E1 -1031.842,E2 -1031.842} C_VEL
LIN {X 0,Y 594.373,Z 387.678,A -85,B 0,C 180,E1 -1033.048,E2 -1033.048} C_VEL
LIN {X 0,Y 594.445,Z 377.969,A -85,B 0,C 180,E1 -1034.229,E2 -1034.229} C_VEL
LIN {X 0,Y 594.505,Z 367.199,A -85,B 0,C 180,E1 -1035.33,E2 -1035.33} C_VEL
LIN {X 0,Y 594.595,Z 356.103,A -85,B 0,C 180,E1 -1036.283,E2 -1036.283} C_VEL
LIN {X 0,Y 594.674,Z 342.72,A -85,B 0,C 180,E1 -1037.247,E2 -1037.247} C_VEL
LIN {X 0,Y 594.77,Z 329.699,A -85,B 0,C 180,E1 -1038.015,E2 -1038.015} C_VEL
LIN {X 0,Y 594.86,Z 316.375,A -85,B 0,C 180,E1 -1038.657,E2 -1038.657} C_VEL
LIN {X 0,Y 594.94,Z 301.883,A -85,B 0,C 180,E1 -1039.207,E2 -1039.207} C_VEL
LIN {X 0,Y 595.024,Z 286.555,A -85,B 0,C 180,E1 -1039.638,E2 -1039.638} C_VEL
LIN {X 0,Y 595.036,Z 273.169,A -85,B 0,C 180,E1 -1039.896,E2 -1039.896} C_VEL
LIN {X 0,Y 594.238,Z 269.367,A -85,B 0,C 180,E1 -1039.993,E2 -1039.993} C_VEL
LIN {X 0,Y 594.215,Z 265.788,A -85,B 0,C 180,E1 -1042.902,E2 -1042.902} C_VEL
LIN {X 0,Y 594.239,Z 262.188,A -85,B 0,C 180,E1 -1045.881,E2 -1045.881} C_VEL
LIN {X 0,Y 594.276,Z 258.915,A -85,B 0,C 180,E1 -1048.646,E2 -1048.646} C_VEL
LIN {X 0,Y 594.248,Z 256.116,A -85,B 0,C 180,E1 -1051.065,E2 -1051.065} C_VEL
LIN {X 0,Y 594.265,Z 253.842,A -85,B 0,C 180,E1 -1053.296,E2 -1053.296} C_VEL
LIN {X 0,Y 594.325,Z 251.586,A -85,B 0,C 180,E1 -1055.578,E2 -1055.578} C_VEL
LIN {X 0,Y 594.286,Z 248.676,A -85,B 0,C 180,E1 -1058.495,E2 -1058.495} C_VEL
LIN {X 0,Y 594.328,Z 246.083,A -85,B 0,C 180,E1 -1061.085,E2 -1061.085} C_VEL
LIN {X 0,Y 594.409,Z 246.073,A -85,B 0,C 180,E1 -1063.516,E2 -1063.516} C_VEL
LIN {X 0,Y 594.379,Z 246.074,A -85,B 0,C 180,E1 -1066.322,E2 -1066.322} C_VEL
LIN {X 0,Y 594.374,Z 246.074,A -85,B 0,C 180,E1 -1069.096,E2 -1069.096} C_VEL
LIN {X 0,Y 594.414,Z 246.071,A -85,B 0,C 180,E1 -1071.844,E2 -1071.844} C_VEL
LIN {X 0,Y 594.388,Z 246.072,A -85,B 0,C 180,E1 -1074.573,E2 -1074.573} C_VEL
LIN {X 0,Y 594.413,Z 246.071,A -85,B 0,C 180,E1 -1077.29,E2 -1077.29} C_VEL
LIN {X 0,Y 594.411,Z 246.069,A -85,B 0,C 180,E1 -1080.001,E2 -1080.001} C_VEL
LIN {X 0,Y 594.41,Z 246.07,A -85,B 0,C 180,E1 -1082.711,E2 -1082.711} C_VEL
LIN {X 0,Y 594.393,Z 246.073,A -85,B 0,C 180,E1 -1085.428,E2 -1085.428} C_VEL
LIN {X 0,Y 594.414,Z 246.069,A -85,B 0,C 180,E1 -1088.157,E2 -1088.157} C_VEL
LIN {X 0,Y 594.388,Z 246.074,A -85,B 0,C 180,E1 -1091.076,E2 -1091.076} C_VEL
LIN {X 0,Y 594.385,Z 246.073,A -85,B 0,C 180,E1 -1093.679,E2 -1093.679} C_VEL
LIN {X 0,Y 594.392,Z 246.071,A -85,B 0,C 180,E1 -1096.721,E2 -1096.721} C_VEL
LIN {X 0,Y 594.366,Z 246.077,A -85,B 0,C 180,E1 -1099.335,E2 -1099.335} C_VEL
LIN {X 0,Y 594.369,Z 246.077,A -85,B 0,C 180,E1 -1101.504,E2 -1101.504} C_VEL
LIN {X 0,Y 594.386,Z 246.074,A -85,B 0,C 180,E1 -1104.447,E2 -1104.447} C_VEL
LIN {X 0,Y 594.388,Z 246.075,A -85,B 0,C 180,E1 -1106.7,E2 -1106.7} C_VEL
LIN {X 0,Y 594.379,Z 246.076,A -85,B 0,C 180,E1 -1108.999,E2 -1108.999} C_VEL
LIN {X 0,Y 594.375,Z 246.075,A -85,B 0,C 180,E1 -1111.643,E2 -1111.643} C_VEL
LIN {X 0,Y 594.383,Z 246.074,A -85,B 0,C 180,E1 -1114.58,E2 -1114.58} C_VEL
LIN {X 0,Y 594.389,Z 246.073,A -85,B 0,C 180,E1 -1117.609,E2 -1117.609} C_VEL
LIN {X 0,Y 594.37,Z 246.077,A -85,B 0,C 180,E1 -1120.567,E2 -1120.567} C_VEL
LIN {X 0,Y 594.364,Z 246.076,A -85,B 0,C 180,E1 -1123.3,E2 -1123.3} C_VEL
LIN {X 0,Y 594.381,Z 246.074,A -85,B 0,C 180,E1 -1126.159,E2 -1126.159} C_VEL
LIN {X 0,Y 594.426,Z 246.204,A -85,B 0,C 180,E1 -1127.92,E2 -1127.92} C_VEL
LIN {X 0,Y 594.691,Z 249.527,A -85,B 0,C 180,E1 -1129.143,E2 -1129.143} C_VEL
LIN {X 0,Y 594.626,Z 256.666,A -85,B 0,C 180,E1 -1131.672,E2 -1131.672} C_VEL
LIN {X 0,Y 594.585,Z 264.022,A -85,B 0,C 180,E1 -1134.191,E2 -1134.191} C_VEL
LIN {X 0,Y 594.543,Z 271.449,A -85,B 0,C 180,E1 -1136.656,E2 -1136.656} C_VEL
LIN {X 0,Y 594.502,Z 278.875,A -85,B 0,C 180,E1 -1139.054,E2 -1139.054} C_VEL
LIN {X 0,Y 594.457,Z 287.54,A -85,B 0,C 180,E1 -1141.778,E2 -1141.778} C_VEL
LIN {X 0,Y 594.435,Z 296.205,A -85,B 0,C 180,E1 -1144.435,E2 -1144.435} C_VEL
LIN {X 0,Y 594.357,Z 305.657,A -85,B 0,C 180,E1 -1147.267,E2 -1147.267} C_VEL
LIN {X 0,Y 594.357,Z 314.772,A -85,B 0,C 180,E1 -1149.946,E2 -1149.946} C_VEL
LIN {X 0,Y 594.303,Z 324.674,A -85,B 0,C 180,E1 -1152.805,E2 -1152.805} C_VEL
LIN {X 0,Y 594.307,Z 325.419,A -85,B 0,C 180,E1 -1153.018,E2 -1153.018} C_VEL
LIN {X 0,Y 595.081,Z 329.893,A -85,B 0,C 180,E1 -1153.102,E2 -1153.102} C_VEL
LIN {X 0,Y 595.061,Z 345.242,A -85,B 0,C 180,E1 -1153.376,E2 -1153.376} C_VEL
LIN {X 0,Y 594.986,Z 359.315,A -85,B 0,C 180,E1 -1153.752,E2 -1153.752} C_VEL
LIN {X 0,Y 594.861,Z 373.805,A -85,B 0,C 180,E1 -1154.277,E2 -1154.277} C_VEL
LIN {X 0,Y 594.759,Z 387.872,A -85,B 0,C 180,E1 -1154.933,E2 -1154.933} C_VEL
LIN {X 0,Y 594.682,Z 401.414,A -85,B 0,C 180,E1 -1155.715,E2 -1155.715} C_VEL
LIN {X 0,Y 594.587,Z 413.861,A -85,B 0,C 180,E1 -1156.588,E2 -1156.588} C_VEL
LIN {X 0,Y 594.535,Z 425.281,A -85,B 0,C 180,E1 -1157.542,E2 -1157.542} C_VEL
LIN {X 0,Y 594.434,Z 435.715,A -85,B 0,C 180,E1 -1158.572,E2 -1158.572} C_VEL
LIN {X 0,Y 594.38,Z 446.024,A -85,B 0,C 180,E1 -1159.784,E2 -1159.784} C_VEL
LIN {X 0,Y 594.337,Z 454.536,A -85,B 0,C 180,E1 -1160.986,E2 -1160.986} C_VEL
LIN {X 0,Y 594.31,Z 461.614,A -85,B 0,C 180,E1 -1162.184,E2 -1162.184} C_VEL
LIN {X 0,Y 594.261,Z 468.495,A -85,B 0,C 180,E1 -1163.624,E2 -1163.624} C_VEL
LIN {X 0,Y 594.245,Z 473.325,A -85,B 0,C 180,E1 -1164.912,E2 -1164.912} C_VEL
LIN {X 0,Y 594.254,Z 476.289,A -85,B 0,C 180,E1 -1165.931,E2 -1165.931} C_VEL
LIN {X 0,Y 594.221,Z 479.186,A -85,B 0,C 180,E1 -1167.289,E2 -1167.289} C_VEL
LIN {X 0,Y 594.244,Z 480.913,A -85,B 0,C 180,E1 -1168.645,E2 -1168.645} C_VEL
LIN {X 0,Y 594.233,Z 481.5,A -85,B 0,C 180,E1 -1170,E2 -1170} C_VEL
LIN {X 0,Y 594.244,Z 480.912,A -85,B 0,C 180,E1 -1171.356,E2 -1171.356} C_VEL
LIN {X 0,Y 594.221,Z 479.184,A -85,B 0,C 180,E1 -1172.712,E2 -1172.712} C_VEL
LIN {X 0,Y 594.254,Z 476.287,A -85,B 0,C 180,E1 -1174.07,E2 -1174.07} C_VEL
LIN {X 0,Y 594.274,Z 472.16,A -85,B 0,C 180,E1 -1175.429,E2 -1175.429} C_VEL
LIN {X 0,Y 594.275,Z 466.701,A -85,B 0,C 180,E1 -1176.792,E2 -1176.792} C_VEL
LIN {X 0,Y 594.323,Z 459.749,A -85,B 0,C 180,E1 -1178.158,E2 -1178.158} C_VEL
LIN {X 0,Y 594.341,Z 451.089,A -85,B 0,C 180,E1 -1179.53,E2 -1179.53} C_VEL
LIN {X 0,Y 594.401,Z 441.873,A -85,B 0,C 180,E1 -1180.733,E2 -1180.733} C_VEL
LIN {X 0,Y 594.468,Z 432.505,A -85,B 0,C 180,E1 -1181.768,E2 -1181.768} C_VEL
LIN {X 0,Y 594.552,Z 421.383,A -85,B 0,C 180,E1 -1182.806,E2 -1182.806} C_VEL
LIN {X 0,Y 594.653,Z 408.638,A -85,B 0,C 180,E1 -1183.799,E2 -1183.799} C_VEL
LIN {X 0,Y 594.739,Z 395.776,A -85,B 0,C 180,E1 -1184.631,E2 -1184.631} C_VEL
LIN {X 0,Y 594.801,Z 382.603,A -85,B 0,C 180,E1 -1185.33,E2 -1185.33} C_VEL
LIN {X 0,Y 594.916,Z 368.173,A -85,B 0,C 180,E1 -1185.942,E2 -1185.942} C_VEL
LIN {X 0,Y 594.998,Z 353.237,A -85,B 0,C 180,E1 -1186.425,E2 -1186.425} C_VEL
LIN {X 0,Y 595.074,Z 338.429,A -85,B 0,C 180,E1 -1186.762,E2 -1186.762} C_VEL
LIN {X 0,Y 594.893,Z 328.251,A -85,B 0,C 180,E1 -1186.927,E2 -1186.927} C_VEL
LIN {X 0,Y 594.308,Z 325.415,A -85,B 0,C 180,E1 -1186.983,E2 -1186.983} C_VEL
LIN {X 0,Y 594.371,Z 316.006,A -85,B 0,C 180,E1 -1189.694,E2 -1189.694} C_VEL
LIN {X 0,Y 594.382,Z 307.341,A -85,B 0,C 180,E1 -1192.233,E2 -1192.233} C_VEL
LIN {X 0,Y 594.386,Z 298.677,A -85,B 0,C 180,E1 -1194.819,E2 -1194.819} C_VEL
LIN {X 0,Y 594.447,Z 289.753,A -85,B 0,C 180,E1 -1197.538,E2 -1197.538} C_VEL
LIN {X 0,Y 594.493,Z 282.585,A -85,B 0,C 180,E1 -1199.77,E2 -1199.77} C_VEL
LIN {X 0,Y 594.465,Z 273.939,A -85,B 0,C 180,E1 -1202.537,E2 -1202.537} C_VEL
LIN {X 0,Y 594.535,Z 266.556,A -85,B 0,C 180,E1 -1204.962,E2 -1204.962} C_VEL
LIN {X 0,Y 594.645,Z 257.829,A -85,B 0,C 180,E1 -1207.922,E2 -1207.922} C_VEL
LIN {X 0,Y 594.66,Z 250.403,A -85,B 0,C 180,E1 -1210.543,E2 -1210.543} C_VEL
LIN {X 0,Y 594.508,Z 246.721,A -85,B 0,C 180,E1 -1211.862,E2 -1211.862} C_VEL
LIN {X 0,Y 594.387,Z 246.073,A -85,B 0,C 180,E1 -1212.157,E2 -1212.157} C_VEL
LIN {X 0,Y 594.36,Z 246.076,A -85,B 0,C 180,E1 -1214.808,E2 -1214.808} C_VEL
LIN {X 0,Y 594.368,Z 246.075,A -85,B 0,C 180,E1 -1217.624,E2 -1217.624} C_VEL
LIN {X 0,Y 594.377,Z 246.075,A -85,B 0,C 180,E1 -1220.319,E2 -1220.319} C_VEL
LIN {X 0,Y 594.388,Z 246.072,A -85,B 0,C 180,E1 -1222.913,E2 -1222.913} C_VEL
LIN {X 0,Y 594.378,Z 246.075,A -85,B 0,C 180,E1 -1225.863,E2 -1225.863} C_VEL
LIN {X 0,Y 594.375,Z 246.075,A -85,B 0,C 180,E1 -1228.65,E2 -1228.65} C_VEL
LIN {X 0,Y 594.382,Z 246.075,A -85,B 0,C 180,E1 -1231.043,E2 -1231.043} C_VEL
LIN {X 0,Y 594.387,Z 246.073,A -85,B 0,C 180,E1 -1233.3,E2 -1233.3} C_VEL
LIN {X 0,Y 594.391,Z 246.074,A -85,B 0,C 180,E1 -1236.296,E2 -1236.296} C_VEL
LIN {X 0,Y 594.407,Z 246.072,A -85,B 0,C 180,E1 -1239.224,E2 -1239.224} C_VEL
LIN {X 0,Y 594.356,Z 246.076,A -85,B 0,C 180,E1 -1242.095,E2 -1242.095} C_VEL
LIN {X 0,Y 594.368,Z 246.075,A -85,B 0,C 180,E1 -1244.219,E2 -1244.219} C_VEL
LIN {X 0,Y 594.378,Z 246.074,A -85,B 0,C 180,E1 -1246.32,E2 -1246.32} C_VEL
LIN {X 0,Y 594.374,Z 246.074,A -85,B 0,C 180,E1 -1249.094,E2 -1249.094} C_VEL
LIN {X 0,Y 594.414,Z 246.072,A -85,B 0,C 180,E1 -1251.843,E2 -1251.843} C_VEL
LIN {X 0,Y 594.4,Z 246.071,A -85,B 0,C 180,E1 -1254.572,E2 -1254.572} C_VEL
LIN {X 0,Y 594.405,Z 246.071,A -85,B 0,C 180,E1 -1257.289,E2 -1257.289} C_VEL
LIN {X 0,Y 594.415,Z 246.07,A -85,B 0,C 180,E1 -1259.999,E2 -1259.999} C_VEL
LIN {X 0,Y 594.412,Z 246.069,A -85,B 0,C 180,E1 -1262.71,E2 -1262.71} C_VEL
LIN {X 0,Y 594.392,Z 246.074,A -85,B 0,C 180,E1 -1265.427,E2 -1265.427} C_VEL
LIN {X 0,Y 594.415,Z 246.069,A -85,B 0,C 180,E1 -1268.156,E2 -1268.156} C_VEL
LIN {X 0,Y 594.393,Z 246.071,A -85,B 0,C 180,E1 -1271.074,E2 -1271.074} C_VEL
LIN {X 0,Y 594.382,Z 246.075,A -85,B 0,C 180,E1 -1273.678,E2 -1273.678} C_VEL
LIN {X 0,Y 594.36,Z 246.075,A -85,B 0,C 180,E1 -1275.326,E2 -1275.326} C_VEL
LIN {X 0,Y 593.69,Z 246.162,A -85,B 0,C 180,E1 -1275.891,E2 -1275.891} C_VEL
LIN {X 0,Y 590.837,Z 246.517,A -85,B 0,C 180,E1 -1276.81,E2 -1276.81} C_VEL
LIN {X 0,Y 588.433,Z 246.816,A -85,B 0,C 180,E1 -1277.548,E2 -1277.548} C_VEL
LIN {X 0,Y 587.405,Z 246.944,A -85,B 0,C 180,E1 -1278.119,E2 -1278.119} C_VEL
LIN {X 0,Y 587.324,Z 246.953,A -85,B 0,C 180,E1 -1278.312,E2 -1278.312} C_VEL
LIN {X 0,Y 587.331,Z 246.954,A -85,B 0,C 180,E1 -1281.036,E2 -1281.036} C_VEL
LIN {X 0,Y 587.323,Z 246.955,A -85,B 0,C 180,E1 -1283.258,E2 -1283.258} C_VEL
LIN {X 0,Y 587.335,Z 246.952,A -85,B 0,C 180,E1 -1285.515,E2 -1285.515} C_VEL
LIN {X 0,Y 587.349,Z 246.949,A -85,B 0,C 180,E1 -1287.816,E2 -1287.816} C_VEL
LIN {X 0,Y 587.337,Z 246.953,A -85,B 0,C 180,E1 -1290.509,E2 -1290.509} C_VEL
LIN {X 0,Y 587.334,Z 246.951,A -85,B 0,C 180,E1 -1293.395,E2 -1293.395} C_VEL
LIN {X 0,Y 587.355,Z 246.95,A -85,B 0,C 180,E1 -1295.894,E2 -1295.894} C_VEL
LIN {X 0,Y 587.331,Z 246.952,A -85,B 0,C 180,E1 -1298.478,E2 -1298.478} C_VEL
LIN {X 0,Y 587.335,Z 246.952,A -85,B 0,C 180,E1 -1301.155,E2 -1301.155} C_VEL
LIN {X 0,Y 587.33,Z 246.954,A -85,B 0,C 180,E1 -1304.113,E2 -1304.113} C_VEL
LIN {X 0,Y 587.33,Z 246.952,A -85,B 0,C 180,E1 -1306.995,E2 -1306.995} C_VEL
LIN {X 0,Y 587.321,Z 246.953,A -85,B 0,C 180,E1 -1309.979,E2 -1309.979} C_VEL
LIN {X 0,Y 587.339,Z 246.953,A -85,B 0,C 180,E1 -1312.391,E2 -1312.391} C_VEL
LIN {X 0,Y 587.341,Z 246.95,A -85,B 0,C 180,E1 -1314.945,E2 -1314.945} C_VEL
LIN {X 0,Y 587.338,Z 246.951,A -85,B 0,C 180,E1 -1317.42,E2 -1317.42} C_VEL
LIN {X 0,Y 587.339,Z 246.953,A -85,B 0,C 180,E1 -1319.83,E2 -1319.83} C_VEL
LIN {X 0,Y 587.344,Z 246.949,A -85,B 0,C 180,E1 -1322.306,E2 -1322.306} C_VEL
LIN {X 0,Y 587.33,Z 246.951,A -85,B 0,C 180,E1 -1324.483,E2 -1324.483} C_VEL
LIN {X 0,Y 587.313,Z 246.956,A -85,B 0,C 180,E1 -1327.129,E2 -1327.129} C_VEL
LIN {X 0,Y 587.327,Z 246.952,A -85,B 0,C 180,E1 -1329.695,E2 -1329.695} C_VEL
LIN {X 0,Y 587.35,Z 246.949,A -85,B 0,C 180,E1 -1332.594,E2 -1332.594} C_VEL
LIN {X 0,Y 587.355,Z 246.949,A -85,B 0,C 180,E1 -1335.738,E2 -1335.738} C_VEL
LIN {X 0,Y 587.352,Z 246.95,A -85,B 0,C 180,E1 -1338.858,E2 -1338.858} C_VEL
LIN {X 0,Y 587.364,Z 246.95,A -85,B 0,C 180,E1 -1341.744,E2 -1341.744} C_VEL
LIN {X 0,Y 587.355,Z 246.948,A -85,B 0,C 180,E1 -1344.507,E2 -1344.507} C_VEL
LIN {X 0,Y 587.245,Z 247.25,A -85,B 0,C 180,E1 -1345.882,E2 -1345.882} C_VEL
LIN {X 0,Y 587.259,Z 250.073,A -85,B 0,C 180,E1 -1348.628,E2 -1348.628} C_VEL
LIN {X 0,Y 587.233,Z 252.866,A -85,B 0,C 180,E1 -1351.371,E2 -1351.371} C_VEL
LIN {X 0,Y 587.16,Z 255.692,A -85,B 0,C 180,E1 -1354.118,E2 -1354.118} C_VEL
LIN {X 0,Y 587.182,Z 258.641,A -85,B 0,C 180,E1 -1356.874,E2 -1356.874} C_VEL
LIN {X 0,Y 587.146,Z 261.869,A -85,B 0,C 180,E1 -1359.646,E2 -1359.646} C_VEL
LIN {X 0,Y 587.129,Z 265.192,A -85,B 0,C 180,E1 -1362.442,E2 -1362.442} C_VEL
LIN {X 0,Y 587.105,Z 268.615,A -85,B 0,C 180,E1 -1365.269,E2 -1365.269} C_VEL
LIN {X 0,Y 587.13,Z 269.374,A -85,B 0,C 180,E1 -1365.891,E2 -1365.891} C_VEL
LIN {X 0,Y 588.264,Z 274.586,A -85,B 0,C 180,E1 -1366.015,E2 -1366.015} C_VEL
LIN {X 0,Y 588.195,Z 289.637,A -85,B 0,C 180,E1 -1366.329,E2 -1366.329} C_VEL
LIN {X 0,Y 588.075,Z 303.194,A -85,B 0,C 180,E1 -1366.734,E2 -1366.734} C_VEL
LIN {X 0,Y 587.905,Z 318.039,A -85,B 0,C 180,E1 -1367.319,E2 -1367.319} C_VEL
LIN {X 0,Y 587.821,Z 331.95,A -85,B 0,C 180,E1 -1368.02,E2 -1368.02} C_VEL
LIN {X 0,Y 587.712,Z 345.127,A -85,B 0,C 180,E1 -1368.836,E2 -1368.836} C_VEL
LIN {X 0,Y 587.595,Z 357.337,A -85,B 0,C 180,E1 -1369.748,E2 -1369.748} C_VEL
LIN {X 0,Y 587.491,Z 369.599,A -85,B 0,C 180,E1 -1370.847,E2 -1370.847} C_VEL
LIN {X 0,Y 587.376,Z 379.948,A -85,B 0,C 180,E1 -1371.956,E2 -1371.956} C_VEL
LIN {X 0,Y 587.304,Z 390.084,A -85,B 0,C 180,E1 -1373.259,E2 -1373.259} C_VEL
LIN {X 0,Y 587.257,Z 398.438,A -85,B 0,C 180,E1 -1374.563,E2 -1374.563} C_VEL
LIN {X 0,Y 587.213,Z 405.141,A -85,B 0,C 180,E1 -1375.837,E2 -1375.837} C_VEL
LIN {X 0,Y 587.174,Z 410.376,A -85,B 0,C 180,E1 -1377.053,E2 -1377.053} C_VEL
LIN {X 0,Y 587.176,Z 414.309,A -85,B 0,C 180,E1 -1378.214,E2 -1378.214} C_VEL
LIN {X 0,Y 587.126,Z 417.419,A -85,B 0,C 180,E1 -1379.391,E2 -1379.391} C_VEL
LIN {X 0,Y 587.138,Z 419.473,A -85,B 0,C 180,E1 -1380.479,E2 -1380.479} C_VEL
LIN {X 0,Y 587.116,Z 421.001,A -85,B 0,C 180,E1 -1381.802,E2 -1381.802} C_VEL
LIN {X 0,Y 587.139,Z 421.424,A -85,B 0,C 180,E1 -1383.409,E2 -1383.409} C_VEL
LIN {X 0,Y 587.131,Z 420.98,A -85,B 0,C 180,E1 -1384.319,E2 -1384.319} C_VEL
LIN {X 0,Y 587.129,Z 418.991,A -85,B 0,C 180,E1 -1385.911,E2 -1385.911} C_VEL
LIN {X 0,Y 587.161,Z 416.223,A -85,B 0,C 180,E1 -1387.189,E2 -1387.189} C_VEL
LIN {X 0,Y 587.154,Z 412.332,A -85,B 0,C 180,E1 -1388.492,E2 -1388.492} C_VEL
LIN {X 0,Y 587.201,Z 406.294,A -85,B 0,C 180,E1 -1390.007,E2 -1390.007} C_VEL
LIN {X 0,Y 587.234,Z 399.223,A -85,B 0,C 180,E1 -1391.393,E2 -1391.393} C_VEL
LIN {X 0,Y 587.307,Z 390.504,A -85,B 0,C 180,E1 -1392.772,E2 -1392.772} C_VEL
LIN {X 0,Y 587.358,Z 381.547,A -85,B 0,C 180,E1 -1393.946,E2 -1393.946} C_VEL
LIN {X 0,Y 587.457,Z 371.008,A -85,B 0,C 180,E1 -1395.104,E2 -1395.104} C_VEL
LIN {X 0,Y 587.571,Z 359.31,A -85,B 0,C 180,E1 -1396.179,E2 -1396.179} C_VEL
LIN {X 0,Y 587.69,Z 346.789,A -85,B 0,C 180,E1 -1397.139,E2 -1397.139} C_VEL
LIN {X 0,Y 587.848,Z 333.655,A -85,B 0,C 180,E1 -1397.973,E2 -1397.973} C_VEL
LIN {X 0,Y 587.954,Z 320.247,A -85,B 0,C 180,E1 -1398.67,E2 -1398.67} C_VEL
LIN {X 0,Y 588.09,Z 306.3,A -85,B 0,C 180,E1 -1399.249,E2 -1399.249} C_VEL
LIN {X 0,Y 588.194,Z 290.667,A -85,B 0,C 180,E1 -1399.736,E2 -1399.736} C_VEL
LIN {X 0,Y 588.289,Z 275.96,A -85,B 0,C 180,E1 -1400.053,E2 -1400.053} C_VEL
LIN {X 0,Y 587.601,Z 271.728,A -85,B 0,C 180,E1 -1400.137,E2 -1400.137} C_VEL
LIN {X 0,Y 587.166,Z 269.381,A -85,B 0,C 180,E1 -1400.193,E2 -1400.193} C_VEL
LIN {X 0,Y 587.139,Z 265.587,A -85,B 0,C 180,E1 -1403.319,E2 -1403.319} C_VEL
LIN {X 0,Y 587.144,Z 262.667,A -85,B 0,C 180,E1 -1405.767,E2 -1405.767} C_VEL
LIN {X 0,Y 587.177,Z 259.789,A -85,B 0,C 180,E1 -1408.222,E2 -1408.222} C_VEL
LIN {X 0,Y 587.16,Z 256.721,A -85,B 0,C 180,E1 -1410.899,E2 -1410.899} C_VEL
LIN {X 0,Y 587.218,Z 253.982,A -85,B 0,C 180,E1 -1413.846,E2 -1413.846} C_VEL
LIN {X 0,Y 587.232,Z 251.821,A -85,B 0,C 180,E1 -1415.99,E2 -1415.99} C_VEL
LIN {X 0,Y 587.236,Z 249.605,A -85,B 0,C 180,E1 -1418.223,E2 -1418.223} C_VEL
LIN {X 0,Y 587.278,Z 246.961,A -85,B 0,C 180,E1 -1420.977,E2 -1420.977} C_VEL
LIN {X 0,Y 587.35,Z 246.951,A -85,B 0,C 180,E1 -1423.312,E2 -1423.312} C_VEL
LIN {X 0,Y 587.355,Z 246.948,A -85,B 0,C 180,E1 -1426.155,E2 -1426.155} C_VEL
LIN {X 0,Y 587.339,Z 246.951,A -85,B 0,C 180,E1 -1428.963,E2 -1428.963} C_VEL
LIN {X 0,Y 587.368,Z 246.948,A -85,B 0,C 180,E1 -1431.746,E2 -1431.746} C_VEL
LIN {X 0,Y 587.354,Z 246.948,A -85,B 0,C 180,E1 -1434.508,E2 -1434.508} C_VEL
LIN {X 0,Y 587.377,Z 246.948,A -85,B 0,C 180,E1 -1437.258,E2 -1437.258} C_VEL
LIN {X 0,Y 587.38,Z 246.945,A -85,B 0,C 180,E1 -1440.001,E2 -1440.001} C_VEL
LIN {X 0,Y 587.375,Z 246.947,A -85,B 0,C 180,E1 -1442.744,E2 -1442.744} C_VEL
LIN {X 0,Y 587.358,Z 246.949,A -85,B 0,C 180,E1 -1445.494,E2 -1445.494} C_VEL
LIN {X 0,Y 587.367,Z 246.946,A -85,B 0,C 180,E1 -1448.256,E2 -1448.256} C_VEL
LIN {X 0,Y 587.345,Z 246.951,A -85,B 0,C 180,E1 -1451.134,E2 -1451.134} C_VEL
LIN {X 0,Y 587.362,Z 246.949,A -85,B 0,C 180,E1 -1454.261,E2 -1454.261} C_VEL
LIN {X 0,Y 587.349,Z 246.95,A -85,B 0,C 180,E1 -1457.407,E2 -1457.407} C_VEL
LIN {X 0,Y 587.331,Z 246.953,A -85,B 0,C 180,E1 -1460.305,E2 -1460.305} C_VEL
LIN {X 0,Y 587.32,Z 246.953,A -85,B 0,C 180,E1 -1463.259,E2 -1463.259} C_VEL
LIN {X 0,Y 587.339,Z 246.951,A -85,B 0,C 180,E1 -1465.517,E2 -1465.517} C_VEL
LIN {X 0,Y 587.346,Z 246.952,A -85,B 0,C 180,E1 -1467.818,E2 -1467.818} C_VEL
LIN {X 0,Y 587.334,Z 246.951,A -85,B 0,C 180,E1 -1470.511,E2 -1470.511} C_VEL
LIN {X 0,Y 587.331,Z 246.953,A -85,B 0,C 180,E1 -1473.397,E2 -1473.397} C_VEL
LIN {X 0,Y 587.291,Z 246.958,A -85,B 0,C 180,E1 -1475.9,E2 -1475.9} C_VEL
LIN {X 0,Y 587.331,Z 246.954,A -85,B 0,C 180,E1 -1478.48,E2 -1478.48} C_VEL
LIN {X 0,Y 587.336,Z 246.951,A -85,B 0,C 180,E1 -1481.157,E2 -1481.157} C_VEL
LIN {X 0,Y 587.324,Z 246.953,A -85,B 0,C 180,E1 -1484.114,E2 -1484.114} C_VEL
LIN {X 0,Y 587.32,Z 246.955,A -85,B 0,C 180,E1 -1486.995,E2 -1486.995} C_VEL
LIN {X 0,Y 587.367,Z 247.074,A -85,B 0,C 180,E1 -1487.637,E2 -1487.637} C_VEL
LIN {X 0,Y 587.75,Z 250.379,A -85,B 0,C 180,E1 -1488.879,E2 -1488.879} C_VEL
LIN {X 0,Y 587.702,Z 257.833,A -85,B 0,C 180,E1 -1491.55,E2 -1491.55} C_VEL
LIN {X 0,Y 587.622,Z 266.123,A -85,B 0,C 180,E1 -1494.418,E2 -1494.418} C_VEL
LIN {X 0,Y 587.559,Z 273.403,A -85,B 0,C 180,E1 -1496.856,E2 -1496.856} C_VEL
LIN {X 0,Y 587.453,Z 281.448,A -85,B 0,C 180,E1 -1499.471,E2 -1499.471} C_VEL
LIN {X 0,Y 587.473,Z 290.016,A -85,B 0,C 180,E1 -1502.189,E2 -1502.189} C_VEL
LIN {X 0,Y 587.389,Z 298.68,A -85,B 0,C 180,E1 -1504.866,E2 -1504.866} C_VEL
LIN {X 0,Y 587.343,Z 307.345,A -85,B 0,C 180,E1 -1507.487,E2 -1507.487} C_VEL
LIN {X 0,Y 587.316,Z 317.247,A -85,B 0,C 180,E1 -1510.425,E2 -1510.425} C_VEL
LIN {X 0,Y 587.253,Z 325.517,A -85,B 0,C 180,E1 -1512.812,E2 -1512.812} C_VEL
LIN {X 0,Y 588.288,Z 331.089,A -85,B 0,C 180,E1 -1512.919,E2 -1512.919} C_VEL
LIN {X 0,Y 588.225,Z 346.554,A -85,B 0,C 180,E1 -1513.21,E2 -1513.21} C_VEL
LIN {X 0,Y 588.136,Z 361.927,A -85,B 0,C 180,E1 -1513.647,E2 -1513.647} C_VEL
LIN {X 0,Y 587.994,Z 374.854,A -85,B 0,C 180,E1 -1514.133,E2 -1514.133} C_VEL
LIN {X 0,Y 587.86,Z 389.537,A -85,B 0,C 180,E1 -1514.84,E2 -1514.84} C_VEL
LIN {X 0,Y 587.756,Z 402.173,A -85,B 0,C 180,E1 -1515.591,E2 -1515.591} C_VEL
LIN {X 0,Y 587.628,Z 415.021,A -85,B 0,C 180,E1 -1516.514,E2 -1516.514} C_VEL
LIN {X 0,Y 587.522,Z 427.197,A -85,B 0,C 180,E1 -1517.566,E2 -1517.566} C_VEL
LIN {X 0,Y 587.424,Z 437.709,A -85,B 0,C 180,E1 -1518.65,E2 -1518.65} C_VEL
LIN {X 0,Y 587.351,Z 447.374,A -85,B 0,C 180,E1 -1519.835,E2 -1519.835} C_VEL
LIN {X 0,Y 587.265,Z 455.657,A -85,B 0,C 180,E1 -1521.05,E2 -1521.05} C_VEL
LIN {X 0,Y 587.229,Z 463.428,A -85,B 0,C 180,E1 -1522.436,E2 -1522.436} C_VEL
LIN {X 0,Y 587.18,Z 469.609,A -85,B 0,C 180,E1 -1523.817,E2 -1523.817} C_VEL
LIN {X 0,Y 587.136,Z 474.385,A -85,B 0,C 180,E1 -1525.194,E2 -1525.194} C_VEL
LIN {X 0,Y 587.18,Z 477.888,A -85,B 0,C 180,E1 -1526.57,E2 -1526.57} C_VEL
LIN {X 0,Y 587.14,Z 480.193,A -85,B 0,C 180,E1 -1527.943,E2 -1527.943} C_VEL
LIN {X 0,Y 587.135,Z 481.35,A -85,B 0,C 180,E1 -1529.315,E2 -1529.315} C_VEL
LIN {X 0,Y 587.135,Z 481.35,A -85,B 0,C 180,E1 -1530.686,E2 -1530.686} C_VEL
LIN {X 0,Y 587.14,Z 480.191,A -85,B 0,C 180,E1 -1532.058,E2 -1532.058} C_VEL
LIN {X 0,Y 587.18,Z 477.885,A -85,B 0,C 180,E1 -1533.431,E2 -1533.431} C_VEL
LIN {X 0,Y 587.136,Z 474.382,A -85,B 0,C 180,E1 -1534.807,E2 -1534.807} C_VEL
LIN {X 0,Y 587.18,Z 469.606,A -85,B 0,C 180,E1 -1536.184,E2 -1536.184} C_VEL
LIN {X 0,Y 587.23,Z 463.423,A -85,B 0,C 180,E1 -1537.565,E2 -1537.565} C_VEL
LIN {X 0,Y 587.266,Z 455.65,A -85,B 0,C 180,E1 -1538.951,E2 -1538.951} C_VEL
LIN {X 0,Y 587.351,Z 447.367,A -85,B 0,C 180,E1 -1540.166,E2 -1540.166} C_VEL
LIN {X 0,Y 587.401,Z 437.391,A -85,B 0,C 180,E1 -1541.386,E2 -1541.386} C_VEL
LIN {X 0,Y 587.522,Z 427.187,A -85,B 0,C 180,E1 -1542.435,E2 -1542.435} C_VEL
LIN {X 0,Y 587.629,Z 415.01,A -85,B 0,C 180,E1 -1543.487,E2 -1543.487} C_VEL
LIN {X 0,Y 587.776,Z 402.046,A -85,B 0,C 180,E1 -1544.417,E2 -1544.417} C_VEL
LIN {X 0,Y 587.853,Z 387.852,A -85,B 0,C 180,E1 -1545.25,E2 -1545.25} C_VEL
LIN {X 0,Y 588.025,Z 373.782,A -85,B 0,C 180,E1 -1545.912,E2 -1545.912} C_VEL
LIN {X 0,Y 588.171,Z 359.288,A -85,B 0,C 180,E1 -1546.442,E2 -1546.442} C_VEL
LIN {X 0,Y 588.26,Z 343.729,A -85,B 0,C 180,E1 -1546.857,E2 -1546.857} C_VEL
LIN {X 0,Y 588.245,Z 329.886,A -85,B 0,C 180,E1 -1547.1,E2 -1547.1} C_VEL
LIN {X 0,Y 587.258,Z 325.377,A -85,B 0,C 180,E1 -1547.204,E2 -1547.204} C_VEL
LIN {X 0,Y 587.324,Z 316.006,A -85,B 0,C 180,E1 -1549.94,E2 -1549.94} C_VEL
LIN {X 0,Y 587.346,Z 307.341,A -85,B 0,C 180,E1 -1552.514,E2 -1552.514} C_VEL
LIN {X 0,Y 587.425,Z 297.439,A -85,B 0,C 180,E1 -1555.513,E2 -1555.513} C_VEL
LIN {X 0,Y 587.457,Z 287.537,A -85,B 0,C 180,E1 -1558.59,E2 -1558.59} C_VEL
LIN {X 0,Y 587.5,Z 278.872,A -85,B 0,C 180,E1 -1561.358,E2 -1561.358} C_VEL
LIN {X 0,Y 587.567,Z 270.207,A -85,B 0,C 180,E1 -1564.207,E2 -1564.207} C_VEL
LIN {X 0,Y 587.673,Z 261.544,A -85,B 0,C 180,E1 -1567.152,E2 -1567.152} C_VEL
LIN {X 0,Y 587.736,Z 253.301,A -85,B 0,C 180,E1 -1570.066,E2 -1570.066} C_VEL
LIN {X 0,Y 587.697,Z 249.031,A -85,B 0,C 180,E1 -1571.583,E2 -1571.583} C_VEL
LIN {X 0,Y 587.338,Z 246.953,A -85,B 0,C 180,E1 -1572.421,E2 -1572.421} C_VEL
LIN {X 0,Y 587.305,Z 246.957,A -85,B 0,C 180,E1 -1575.087,E2 -1575.087} C_VEL
LIN {X 0,Y 587.325,Z 246.952,A -85,B 0,C 180,E1 -1577.925,E2 -1577.925} C_VEL
LIN {X 0,Y 587.337,Z 246.952,A -85,B 0,C 180,E1 -1580.64,E2 -1580.64} C_VEL
LIN {X 0,Y 587.353,Z 246.949,A -85,B 0,C 180,E1 -1583.292,E2 -1583.292} C_VEL
LIN {X 0,Y 587.341,Z 246.952,A -85,B 0,C 180,E1 -1585.778,E2 -1585.778} C_VEL
LIN {X 0,Y 587.346,Z 246.949,A -85,B 0,C 180,E1 -1588.231,E2 -1588.231} C_VEL
LIN {X 0,Y 587.35,Z 246.951,A -85,B 0,C 180,E1 -1590.867,E2 -1590.867} C_VEL
LIN {X 0,Y 587.342,Z 246.95,A -85,B 0,C 180,E1 -1593.721,E2 -1593.721} C_VEL
LIN {X 0,Y 587.34,Z 246.951,A -85,B 0,C 180,E1 -1595.993,E2 -1595.993} C_VEL
LIN {X 0,Y 587.321,Z 246.955,A -85,B 0,C 180,E1 -1598.225,E2 -1598.225} C_VEL
LIN {X 0,Y 587.356,Z 246.949,A -85,B 0,C 180,E1 -1601.151,E2 -1601.151} C_VEL
LIN {X 0,Y 587.326,Z 246.952,A -85,B 0,C 180,E1 -1604.024,E2 -1604.024} C_VEL
LIN {X 0,Y 587.355,Z 246.948,A -85,B 0,C 180,E1 -1606.154,E2 -1606.154} C_VEL
LIN {X 0,Y 587.342,Z 246.95,A -85,B 0,C 180,E1 -1608.962,E2 -1608.962} C_VEL
LIN {X 0,Y 587.367,Z 246.949,A -85,B 0,C 180,E1 -1611.744,E2 -1611.744} C_VEL
LIN {X 0,Y 587.364,Z 246.947,A -85,B 0,C 180,E1 -1614.506,E2 -1614.506} C_VEL
LIN {X 0,Y 587.373,Z 246.947,A -85,B 0,C 180,E1 -1617.256,E2 -1617.256} C_VEL
LIN {X 0,Y 587.384,Z 246.946,A -85,B 0,C 180,E1 -1619.999,E2 -1619.999} C_VEL
LIN {X 0,Y 587.378,Z 246.945,A -85,B 0,C 180,E1 -1622.742,E2 -1622.742} C_VEL
LIN {X 0,Y 587.357,Z 246.95,A -85,B 0,C 180,E1 -1625.492,E2 -1625.492} C_VEL
LIN {X 0,Y 587.368,Z 246.947,A -85,B 0,C 180,E1 -1628.254,E2 -1628.254} C_VEL
LIN {X 0,Y 587.351,Z 246.948,A -85,B 0,C 180,E1 -1631.133,E2 -1631.133} C_VEL
LIN {X 0,Y 587.368,Z 246.947,A -85,B 0,C 180,E1 -1634.26,E2 -1634.26} C_VEL
LIN {X 0,Y 587.358,Z 246.948,A -85,B 0,C 180,E1 -1637.405,E2 -1637.405} C_VEL
LIN {X 0,Y 587.324,Z 246.953,A -85,B 0,C 180,E1 -1638.312,E2 -1638.312} C_VEL
LIN {X 0,Y 586.671,Z 247.035,A -85,B 0,C 180,E1 -1638.883,E2 -1638.883} C_VEL
LIN {X 0,Y 583.839,Z 247.389,A -85,B 0,C 180,E1 -1639.812,E2 -1639.812} C_VEL
LIN {X 0,Y 581.43,Z 247.69,A -85,B 0,C 180,E1 -1640.559,E2 -1640.559} C_VEL
LIN {X 0,Y 580.378,Z 247.819,A -85,B 0,C 180,E1 -1641.135,E2 -1641.135} C_VEL
LIN {X 0,Y 580.283,Z 247.83,A -85,B 0,C 180,E1 -1641.33,E2 -1641.33} C_VEL
LIN {X 0,Y 580.301,Z 247.829,A -85,B 0,C 180,E1 -1644.315,E2 -1644.315} C_VEL
LIN {X 0,Y 580.276,Z 247.83,A -85,B 0,C 180,E1 -1646.622,E2 -1646.622} C_VEL
LIN {X 0,Y 580.302,Z 247.828,A -85,B 0,C 180,E1 -1649.309,E2 -1649.309} C_VEL
LIN {X 0,Y 580.3,Z 247.827,A -85,B 0,C 180,E1 -1652.199,E2 -1652.199} C_VEL
LIN {X 0,Y 580.3,Z 247.829,A -85,B 0,C 180,E1 -1654.694,E2 -1654.694} C_VEL
LIN {X 0,Y 580.297,Z 247.827,A -85,B 0,C 180,E1 -1657.267,E2 -1657.267} C_VEL
LIN {X 0,Y 580.294,Z 247.828,A -85,B 0,C 180,E1 -1660.27,E2 -1660.27} C_VEL
LIN {X 0,Y 580.277,Z 247.83,A -85,B 0,C 180,E1 -1662.705,E2 -1662.705} C_VEL
LIN {X 0,Y 580.269,Z 247.831,A -85,B 0,C 180,E1 -1665.607,E2 -1665.607} C_VEL
LIN {X 0,Y 580.309,Z 247.829,A -85,B 0,C 180,E1 -1668.233,E2 -1668.233} C_VEL
LIN {X 0,Y 580.283,Z 247.829,A -85,B 0,C 180,E1 -1670.965,E2 -1670.965} C_VEL
LIN {X 0,Y 580.29,Z 247.831,A -85,B 0,C 180,E1 -1673.597,E2 -1673.597} C_VEL
LIN {X 0,Y 580.312,Z 247.826,A -85,B 0,C 180,E1 -1676.145,E2 -1676.145} C_VEL
LIN {X 0,Y 580.286,Z 247.831,A -85,B 0,C 180,E1 -1678.615,E2 -1678.615} C_VEL
LIN {X 0,Y 580.29,Z 247.83,A -85,B 0,C 180,E1 -1681.023,E2 -1681.023} C_VEL
LIN {X 0,Y 580.32,Z 247.825,A -85,B 0,C 180,E1 -1683.657,E2 -1683.657} C_VEL
LIN {X 0,Y 580.275,Z 247.83,A -85,B 0,C 180,E1 -1686.441,E2 -1686.441} C_VEL
LIN {X 0,Y 580.276,Z 247.831,A -85,B 0,C 180,E1 -1689.437,E2 -1689.437} C_VEL
LIN {X 0,Y 580.273,Z 247.831,A -85,B 0,C 180,E1 -1691.645,E2 -1691.645} C_VEL
LIN {X 0,Y 580.273,Z 247.83,A -85,B 0,C 180,E1 -1693.825,E2 -1693.825} C_VEL
LIN {X 0,Y 580.273,Z 247.832,A -85,B 0,C 180,E1 -1696.695,E2 -1696.695} C_VEL
LIN {X 0,Y 580.299,Z 247.829,A -85,B 0,C 180,E1 -1699.533,E2 -1699.533} C_VEL
LIN {X 0,Y 580.332,Z 247.823,A -85,B 0,C 180,E1 -1702.344,E2 -1702.344} C_VEL
LIN {X 0,Y 580.275,Z 247.833,A -85,B 0,C 180,E1 -1705.136,E2 -1705.136} C_VEL
LIN {X 0,Y 580.196,Z 247.85,A -85,B 0,C 180,E1 -1705.832,E2 -1705.832} C_VEL
LIN {X 0,Y 580.199,Z 250.672,A -85,B 0,C 180,E1 -1708.611,E2 -1708.611} C_VEL
LIN {X 0,Y 580.171,Z 253.483,A -85,B 0,C 180,E1 -1711.388,E2 -1711.388} C_VEL
LIN {X 0,Y 580.097,Z 256.322,A -85,B 0,C 180,E1 -1714.168,E2 -1714.168} C_VEL
LIN {X 0,Y 580.111,Z 259.126,A -85,B 0,C 180,E1 -1716.958,E2 -1716.958} C_VEL
LIN {X 0,Y 580.047,Z 262.36,A -85,B 0,C 180,E1 -1719.766,E2 -1719.766} C_VEL
LIN {X 0,Y 580.041,Z 265.687,A -85,B 0,C 180,E1 -1722.597,E2 -1722.597} C_VEL
LIN {X 0,Y 580.03,Z 269.115,A -85,B 0,C 180,E1 -1725.459,E2 -1725.459} C_VEL
LIN {X 0,Y 580.034,Z 269.387,A -85,B 0,C 180,E1 -1725.685,E2 -1725.685} C_VEL
LIN {X 0,Y 581.503,Z 276.721,A -85,B 0,C 180,E1 -1725.846,E2 -1725.846} C_VEL
LIN {X 0,Y 581.362,Z 292.025,A -85,B 0,C 180,E1 -1726.188,E2 -1726.188} C_VEL
LIN {X 0,Y 581.19,Z 307.512,A -85,B 0,C 180,E1 -1726.69,E2 -1726.69} C_VEL
LIN {X 0,Y 581.053,Z 321.832,A -85,B 0,C 180,E1 -1727.304,E2 -1727.304} C_VEL
LIN {X 0,Y 580.913,Z 335.805,A -85,B 0,C 180,E1 -1728.06,E2 -1728.06} C_VEL
LIN {X 0,Y 580.759,Z 349.579,A -85,B 0,C 180,E1 -1728.979,E2 -1728.979} C_VEL
LIN {X 0,Y 580.572,Z 362.161,A -85,B 0,C 180,E1 -1729.997,E2 -1729.997} C_VEL
LIN {X 0,Y 580.431,Z 373.674,A -85,B 0,C 180,E1 -1731.116,E2 -1731.116} C_VEL
LIN {X 0,Y 580.35,Z 383.38,A -85,B 0,C 180,E1 -1732.236,E2 -1732.236} C_VEL
LIN {X 0,Y 580.236,Z 391.926,A -85,B 0,C 180,E1 -1733.402,E2 -1733.402} C_VEL
LIN {X 0,Y 580.186,Z 399.849,A -85,B 0,C 180,E1 -1734.704,E2 -1734.704} C_VEL
LIN {X 0,Y 580.116,Z 406.675,A -85,B 0,C 180,E1 -1736.081,E2 -1736.081} C_VEL
LIN {X 0,Y 580.084,Z 411.909,A -85,B 0,C 180,E1 -1737.412,E2 -1737.412} C_VEL
LIN {X 0,Y 580.071,Z 415.562,A -85,B 0,C 180,E1 -1738.592,E2 -1738.592} C_VEL
LIN {X 0,Y 580.037,Z 418.329,A -85,B 0,C 180,E1 -1739.786,E2 -1739.786} C_VEL
LIN {X 0,Y 580.048,Z 419.805,A -85,B 0,C 180,E1 -1740.658,E2 -1740.658} C_VEL
LIN {X 0,Y 580.024,Z 421.29,A -85,B 0,C 180,E1 -1742.217,E2 -1742.217} C_VEL
LIN {X 0,Y 580.049,Z 421.453,A -85,B 0,C 180,E1 -1743.28,E2 -1743.28} C_VEL
LIN {X 0,Y 580.035,Z 420.661,A -85,B 0,C 180,E1 -1744.713,E2 -1744.713} C_VEL
LIN {X 0,Y 580.028,Z 419.337,A -85,B 0,C 180,E1 -1745.729,E2 -1745.729} C_VEL
LIN {X 0,Y 580.061,Z 416.107,A -85,B 0,C 180,E1 -1747.286,E2 -1747.286} C_VEL
LIN {X 0,Y 580.079,Z 412.17,A -85,B 0,C 180,E1 -1748.605,E2 -1748.605} C_VEL
LIN {X 0,Y 580.113,Z 406.963,A -85,B 0,C 180,E1 -1749.947,E2 -1749.947} C_VEL
LIN {X 0,Y 580.156,Z 400.229,A -85,B 0,C 180,E1 -1751.319,E2 -1751.319} C_VEL
LIN {X 0,Y 580.236,Z 391.78,A -85,B 0,C 180,E1 -1752.709,E2 -1752.709} C_VEL
LIN {X 0,Y 580.343,Z 383.092,A -85,B 0,C 180,E1 -1753.891,E2 -1753.891} C_VEL
LIN {X 0,Y 580.442,Z 372.541,A -85,B 0,C 180,E1 -1755.097,E2 -1755.097} C_VEL
LIN {X 0,Y 580.592,Z 360.337,A -85,B 0,C 180,E1 -1756.253,E2 -1756.253} C_VEL
LIN {X 0,Y 580.751,Z 348.087,A -85,B 0,C 180,E1 -1757.22,E2 -1757.22} C_VEL
LIN {X 0,Y 580.937,Z 335.334,A -85,B 0,C 180,E1 -1758.058,E2 -1758.058} C_VEL
LIN {X 0,Y 581.09,Z 320.685,A -85,B 0,C 180,E1 -1758.84,E2 -1758.84} C_VEL
LIN {X 0,Y 581.247,Z 306.728,A -85,B 0,C 180,E1 -1759.429,E2 -1759.429} C_VEL
LIN {X 0,Y 581.4,Z 291.302,A -85,B 0,C 180,E1 -1759.921,E2 -1759.921} C_VEL
LIN {X 0,Y 581.431,Z 275.438,A -85,B 0,C 180,E1 -1760.268,E2 -1760.268} C_VEL
LIN {X 0,Y 580.052,Z 269.369,A -85,B 0,C 180,E1 -1760.42,E2 -1760.42} C_VEL
LIN {X 0,Y 580.037,Z 266.156,A -85,B 0,C 180,E1 -1763.099,E2 -1763.099} C_VEL
LIN {X 0,Y 580.052,Z 263.35,A -85,B 0,C 180,E1 -1765.476,E2 -1765.476} C_VEL
LIN {X 0,Y 580.064,Z 260.416,A -85,B 0,C 180,E1 -1768.006,E2 -1768.006} C_VEL
LIN {X 0,Y 580.092,Z 258.029,A -85,B 0,C 180,E1 -1770.218,E2 -1770.218} C_VEL
LIN {X 0,Y 580.118,Z 255.904,A -85,B 0,C 180,E1 -1772.591,E2 -1772.591} C_VEL
LIN {X 0,Y 580.183,Z 253.164,A -85,B 0,C 180,E1 -1775.298,E2 -1775.298} C_VEL
LIN {X 0,Y 580.182,Z 250.529,A -85,B 0,C 180,E1 -1777.945,E2 -1777.945} C_VEL
LIN {X 0,Y 580.161,Z 248.323,A -85,B 0,C 180,E1 -1780.174,E2 -1780.174} C_VEL
LIN {X 0,Y 580.218,Z 247.841,A -85,B 0,C 180,E1 -1780.912,E2 -1780.912} C_VEL
LIN {X 0,Y 580.324,Z 247.825,A -85,B 0,C 180,E1 -1783.104,E2 -1783.104} C_VEL
LIN {X 0,Y 580.321,Z 247.825,A -85,B 0,C 180,E1 -1785.984,E2 -1785.984} C_VEL
LIN {X 0,Y 580.298,Z 247.83,A -85,B 0,C 180,E1 -1788.828,E2 -1788.828} C_VEL
LIN {X 0,Y 580.331,Z 247.824,A -85,B 0,C 180,E1 -1791.645,E2 -1791.645} C_VEL
LIN {X 0,Y 580.321,Z 247.825,A -85,B 0,C 180,E1 -1794.441,E2 -1794.441} C_VEL
LIN {X 0,Y 580.342,Z 247.824,A -85,B 0,C 180,E1 -1797.224,E2 -1797.224} C_VEL
LIN {X 0,Y 580.349,Z 247.821,A -85,B 0,C 180,E1 -1800.001,E2 -1800.001} C_VEL
LIN {X 0,Y 580.341,Z 247.823,A -85,B 0,C 180,E1 -1802.777,E2 -1802.777} C_VEL
LIN {X 0,Y 580.323,Z 247.826,A -85,B 0,C 180,E1 -1805.56,E2 -1805.56} C_VEL
LIN {X 0,Y 580.331,Z 247.823,A -85,B 0,C 180,E1 -1808.357,E2 -1808.357} C_VEL
LIN {X 0,Y 580.296,Z 247.828,A -85,B 0,C 180,E1 -1811.192,E2 -1811.192} C_VEL
LIN {X 0,Y 580.325,Z 247.826,A -85,B 0,C 180,E1 -1814.018,E2 -1814.018} C_VEL
LIN {X 0,Y 580.309,Z 247.826,A -85,B 0,C 180,E1 -1816.914,E2 -1816.914} C_VEL
LIN {X 0,Y 580.304,Z 247.826,A -85,B 0,C 180,E1 -1819.823,E2 -1819.823} C_VEL
LIN {X 0,Y 580.273,Z 247.83,A -85,B 0,C 180,E1 -1822.053,E2 -1822.053} C_VEL
LIN {X 0,Y 580.308,Z 247.826,A -85,B 0,C 180,E1 -1825.08,E2 -1825.08} C_VEL
LIN {X 0,Y 580.297,Z 247.831,A -85,B 0,C 180,E1 -1827.86,E2 -1827.86} C_VEL
LIN {X 0,Y 580.282,Z 247.83,A -85,B 0,C 180,E1 -1830.695,E2 -1830.695} C_VEL
LIN {X 0,Y 580.3,Z 247.829,A -85,B 0,C 180,E1 -1833.317,E2 -1833.317} C_VEL
LIN {X 0,Y 580.245,Z 247.835,A -85,B 0,C 180,E1 -1835.757,E2 -1835.757} C_VEL
LIN {X 0,Y 580.287,Z 247.831,A -85,B 0,C 180,E1 -1838.147,E2 -1838.147} C_VEL
LIN {X 0,Y 580.299,Z 247.828,A -85,B 0,C 180,E1 -1840.844,E2 -1840.844} C_VEL
LIN {X 0,Y 580.277,Z 247.833,A -85,B 0,C 180,E1 -1843.658,E2 -1843.658} C_VEL
LIN {X 0,Y 580.284,Z 247.832,A -85,B 0,C 180,E1 -1846.609,E2 -1846.609} C_VEL
LIN {X 0,Y 580.339,Z 247.966,A -85,B 0,C 180,E1 -1847.38,E2 -1847.38} C_VEL
LIN {X 0,Y 580.799,Z 251.23,A -85,B 0,C 180,E1 -1848.611,E2 -1848.611} C_VEL
LIN {X 0,Y 580.782,Z 257.833,A -85,B 0,C 180,E1 -1851.006,E2 -1851.006} C_VEL
LIN {X 0,Y 580.679,Z 265.26,A -85,B 0,C 180,E1 -1853.627,E2 -1853.627} C_VEL
LIN {X 0,Y 580.593,Z 274.103,A -85,B 0,C 180,E1 -1856.641,E2 -1856.641} C_VEL
LIN {X 0,Y 580.456,Z 282.589,A -85,B 0,C 180,E1 -1859.435,E2 -1859.435} C_VEL
LIN {X 0,Y 580.478,Z 290.908,A -85,B 0,C 180,E1 -1862.108,E2 -1862.108} C_VEL
LIN {X 0,Y 580.351,Z 299.918,A -85,B 0,C 180,E1 -1864.923,E2 -1864.923} C_VEL
LIN {X 0,Y 580.306,Z 308.583,A -85,B 0,C 180,E1 -1867.575,E2 -1867.575} C_VEL
LIN {X 0,Y 580.263,Z 317.247,A -85,B 0,C 180,E1 -1870.177,E2 -1870.177} C_VEL
LIN {X 0,Y 580.225,Z 325.385,A -85,B 0,C 180,E1 -1872.583,E2 -1872.583} C_VEL
LIN {X 0,Y 581.476,Z 331.173,A -85,B 0,C 180,E1 -1872.714,E2 -1872.714} C_VEL
LIN {X 0,Y 581.442,Z 346.606,A -85,B 0,C 180,E1 -1873.009,E2 -1873.009} C_VEL
LIN {X 0,Y 581.345,Z 360.629,A -85,B 0,C 180,E1 -1873.405,E2 -1873.405} C_VEL
LIN {X 0,Y 581.167,Z 374.853,A -85,B 0,C 180,E1 -1873.942,E2 -1873.942} C_VEL
LIN {X 0,Y 580.992,Z 389.536,A -85,B 0,C 180,E1 -1874.657,E2 -1874.657} C_VEL
LIN {X 0,Y 580.834,Z 402.886,A -85,B 0,C 180,E1 -1875.464,E2 -1875.464} C_VEL
LIN {X 0,Y 580.677,Z 415.021,A -85,B 0,C 180,E1 -1876.349,E2 -1876.349} C_VEL
LIN {X 0,Y 580.54,Z 427.197,A -85,B 0,C 180,E1 -1877.414,E2 -1877.414} C_VEL
LIN {X 0,Y 580.385,Z 437.709,A -85,B 0,C 180,E1 -1878.511,E2 -1878.511} C_VEL
LIN {X 0,Y 580.308,Z 447.374,A -85,B 0,C 180,E1 -1879.71,E2 -1879.71} C_VEL
LIN {X 0,Y 580.206,Z 455.656,A -85,B 0,C 180,E1 -1880.941,E2 -1880.941} C_VEL
LIN {X 0,Y 580.165,Z 463.428,A -85,B 0,C 180,E1 -1882.343,E2 -1882.343} C_VEL
LIN {X 0,Y 580.094,Z 469.609,A -85,B 0,C 180,E1 -1883.741,E2 -1883.741} C_VEL
LIN {X 0,Y 580.041,Z 474.385,A -85,B 0,C 180,E1 -1885.135,E2 -1885.135} C_VEL
LIN {X 0,Y 580.105,Z 477.888,A -85,B 0,C 180,E1 -1886.528,E2 -1886.528} C_VEL
LIN {X 0,Y 580.039,Z 480.193,A -85,B 0,C 180,E1 -1887.917,E2 -1887.917} C_VEL
LIN {X 0,Y 580.036,Z 481.35,A -85,B 0,C 180,E1 -1889.306,E2 -1889.306} C_VEL
LIN {X 0,Y 580.036,Z 481.35,A -85,B 0,C 180,E1 -1890.695,E2 -1890.695} C_VEL
LIN {X 0,Y 580.039,Z 480.192,A -85,B 0,C 180,E1 -1892.084,E2 -1892.084} C_VEL
LIN {X 0,Y 580.105,Z 477.885,A -85,B 0,C 180,E1 -1893.473,E2 -1893.473} C_VEL
LIN {X 0,Y 580.041,Z 474.382,A -85,B 0,C 180,E1 -1894.866,E2 -1894.866} C_VEL
LIN {X 0,Y 580.093,Z 469.606,A -85,B 0,C 180,E1 -1896.26,E2 -1896.26} C_VEL
LIN {X 0,Y 580.166,Z 463.422,A -85,B 0,C 180,E1 -1897.658,E2 -1897.658} C_VEL
LIN {X 0,Y 580.207,Z 455.649,A -85,B 0,C 180,E1 -1899.06,E2 -1899.06} C_VEL
LIN {X 0,Y 580.309,Z 447.366,A -85,B 0,C 180,E1 -1900.291,E2 -1900.291} C_VEL
LIN {X 0,Y 580.384,Z 437.391,A -85,B 0,C 180,E1 -1901.525,E2 -1901.525} C_VEL
LIN {X 0,Y 580.541,Z 427.187,A -85,B 0,C 180,E1 -1902.587,E2 -1902.587} C_VEL
LIN {X 0,Y 580.675,Z 415.011,A -85,B 0,C 180,E1 -1903.652,E2 -1903.652} C_VEL
LIN {X 0,Y 580.848,Z 402.805,A -85,B 0,C 180,E1 -1904.542,E2 -1904.542} C_VEL
LIN {X 0,Y 580.961,Z 389.517,A -85,B 0,C 180,E1 -1905.345,E2 -1905.345} C_VEL
LIN {X 0,Y 581.168,Z 374.831,A -85,B 0,C 180,E1 -1906.059,E2 -1906.059} C_VEL
LIN {X 0,Y 581.343,Z 360.604,A -85,B 0,C 180,E1 -1906.596,E2 -1906.596} C_VEL
LIN {X 0,Y 581.471,Z 345.719,A -85,B 0,C 180,E1 -1907.012,E2 -1907.012} C_VEL
LIN {X 0,Y 581.375,Z 330.741,A -85,B 0,C 180,E1 -1907.296,E2 -1907.296} C_VEL
LIN {X 0,Y 580.208,Z 325.394,A -85,B 0,C 180,E1 -1907.415,E2 -1907.415} C_VEL
LIN {X 0,Y 580.263,Z 316.006,A -85,B 0,C 180,E1 -1910.194,E2 -1910.194} C_VEL
LIN {X 0,Y 580.297,Z 307.341,A -85,B 0,C 180,E1 -1912.803,E2 -1912.803} C_VEL
LIN {X 0,Y 580.389,Z 298.677,A -85,B 0,C 180,E1 -1915.46,E2 -1915.46} C_VEL
LIN {X 0,Y 580.462,Z 288.774,A -85,B 0,C 180,E1 -1918.572,E2 -1918.572} C_VEL
LIN {X 0,Y 580.524,Z 280.11,A -85,B 0,C 180,E1 -1921.371,E2 -1921.371} C_VEL
LIN {X 0,Y 580.602,Z 271.556,A -85,B 0,C 180,E1 -1924.217,E2 -1924.217} C_VEL
LIN {X 0,Y 580.73,Z 263.481,A -85,B 0,C 180,E1 -1926.991,E2 -1926.991} C_VEL
LIN {X 0,Y 580.806,Z 255.299,A -85,B 0,C 180,E1 -1929.891,E2 -1929.891} C_VEL
LIN {X 0,Y 580.7,Z 250.188,A -85,B 0,C 180,E1 -1931.732,E2 -1931.732} C_VEL
LIN {X 0,Y 580.304,Z 247.829,A -85,B 0,C 180,E1 -1932.704,E2 -1932.704} C_VEL
LIN {X 0,Y 580.262,Z 247.832,A -85,B 0,C 180,E1 -1935.61,E2 -1935.61} C_VEL
LIN {X 0,Y 580.283,Z 247.831,A -85,B 0,C 180,E1 -1938.231,E2 -1938.231} C_VEL
LIN {X 0,Y 580.283,Z 247.829,A -85,B 0,C 180,E1 -1940.965,E2 -1940.965} C_VEL
LIN {X 0,Y 580.273,Z 247.833,A -85,B 0,C 180,E1 -1943.596,E2 -1943.596} C_VEL
LIN {X 0,Y 580.305,Z 247.826,A -85,B 0,C 180,E1 -1946.144,E2 -1946.144} C_VEL
LIN {X 0,Y 580.281,Z 247.83,A -85,B 0,C 180,E1 -1948.614,E2 -1948.614} C_VEL
LIN {X 0,Y 580.293,Z 247.83,A -85,B 0,C 180,E1 -1951.023,E2 -1951.023} C_VEL
LIN {X 0,Y 580.295,Z 247.828,A -85,B 0,C 180,E1 -1953.666,E2 -1953.666} C_VEL
LIN {X 0,Y 580.305,Z 247.826,A -85,B 0,C 180,E1 -1955.683,E2 -1955.683} C_VEL
LIN {X 0,Y 580.273,Z 247.83,A -85,B 0,C 180,E1 -1957.947,E2 -1957.947} C_VEL
LIN {X 0,Y 580.325,Z 247.824,A -85,B 0,C 180,E1 -1960.914,E2 -1960.914} C_VEL
LIN {X 0,Y 580.281,Z 247.83,A -85,B 0,C 180,E1 -1963.825,E2 -1963.825} C_VEL
LIN {X 0,Y 580.323,Z 247.824,A -85,B 0,C 180,E1 -1965.982,E2 -1965.982} C_VEL
LIN {X 0,Y 580.311,Z 247.827,A -85,B 0,C 180,E1 -1968.826,E2 -1968.826} C_VEL
LIN {X 0,Y 580.331,Z 247.824,A -85,B 0,C 180,E1 -1971.643,E2 -1971.643} C_VEL
LIN {X 0,Y 580.328,Z 247.824,A -85,B 0,C 180,E1 -1974.44,E2 -1974.44} C_VEL
LIN {X 0,Y 580.34,Z 247.823,A -85,B 0,C 180,E1 -1977.223,E2 -1977.223} C_VEL
LIN {X 0,Y 580.354,Z 247.821,A -85,B 0,C 180,E1 -1979.999,E2 -1979.999} C_VEL
LIN {X 0,Y 580.344,Z 247.822,A -85,B 0,C 180,E1 -1982.776,E2 -1982.776} C_VEL
LIN {X 0,Y 580.323,Z 247.826,A -85,B 0,C 180,E1 -1985.559,E2 -1985.559} C_VEL
LIN {X 0,Y 580.331,Z 247.825,A -85,B 0,C 180,E1 -1988.355,E2 -1988.355} C_VEL
LIN {X 0,Y 580.303,Z 247.826,A -85,B 0,C 180,E1 -1991.19,E2 -1991.19} C_VEL
LIN {X 0,Y 580.328,Z 247.825,A -85,B 0,C 180,E1 -1994.016,E2 -1994.016} C_VEL
LIN {X 0,Y 580.314,Z 247.827,A -85,B 0,C 180,E1 -1996.913,E2 -1996.913} C_VEL
LIN {X 0,Y 580.288,Z 247.829,A -85,B 0,C 180,E1 -1999.822,E2 -1999.822} C_VEL
LIN {X 0,Y 580.283,Z 247.83,A -85,B 0,C 180,E1 -2001.33,E2 -2001.33} C_VEL
LIN {X 0,Y 579.587,Z 247.918,A -85,B 0,C 180,E1 -2001.909,E2 -2001.909} C_VEL
LIN {X 0,Y 576.71,Z 248.275,A -85,B 0,C 180,E1 -2002.849,E2 -2002.849} C_VEL
LIN {X 0,Y 574.316,Z 248.573,A -85,B 0,C 180,E1 -2003.605,E2 -2003.605} C_VEL
LIN {X 0,Y 573.317,Z 248.699,A -85,B 0,C 180,E1 -2004.189,E2 -2004.189} C_VEL
LIN {X 0,Y 573.25,Z 248.704,A -85,B 0,C 180,E1 -2004.387,E2 -2004.387} C_VEL
LIN {X 0,Y 573.25,Z 248.705,A -85,B 0,C 180,E1 -2006.975,E2 -2006.975} C_VEL
LIN {X 0,Y 573.248,Z 248.708,A -85,B 0,C 180,E1 -2009.488,E2 -2009.488} C_VEL
LIN {X 0,Y 573.254,Z 248.706,A -85,B 0,C 180,E1 -2012.644,E2 -2012.644} C_VEL
LIN {X 0,Y 573.267,Z 248.703,A -85,B 0,C 180,E1 -2015.182,E2 -2015.182} C_VEL
LIN {X 0,Y 573.234,Z 248.71,A -85,B 0,C 180,E1 -2017.806,E2 -2017.806} C_VEL
LIN {X 0,Y 573.266,Z 248.703,A -85,B 0,C 180,E1 -2020.527,E2 -2020.527} C_VEL
LIN {X 0,Y 573.248,Z 248.706,A -85,B 0,C 180,E1 -2023.669,E2 -2023.669} C_VEL
LIN {X 0,Y 573.247,Z 248.705,A -85,B 0,C 180,E1 -2026.641,E2 -2026.641} C_VEL
LIN {X 0,Y 573.268,Z 248.705,A -85,B 0,C 180,E1 -2029.476,E2 -2029.476} C_VEL
LIN {X 0,Y 573.231,Z 248.709,A -85,B 0,C 180,E1 -2032.192,E2 -2032.192} C_VEL
LIN {X 0,Y 573.261,Z 248.704,A -85,B 0,C 180,E1 -2034.815,E2 -2034.815} C_VEL
LIN {X 0,Y 573.251,Z 248.705,A -85,B 0,C 180,E1 -2037.354,E2 -2037.354} C_VEL
LIN {X 0,Y 573.25,Z 248.708,A -85,B 0,C 180,E1 -2039.824,E2 -2039.824} C_VEL
LIN {X 0,Y 573.282,Z 248.701,A -85,B 0,C 180,E1 -2042.234,E2 -2042.234} C_VEL
LIN {X 0,Y 573.26,Z 248.706,A -85,B 0,C 180,E1 -2045.12,E2 -2045.12} C_VEL
LIN {X 0,Y 573.23,Z 248.708,A -85,B 0,C 180,E1 -2047.662,E2 -2047.662} C_VEL
LIN {X 0,Y 573.249,Z 248.706,A -85,B 0,C 180,E1 -2049.923,E2 -2049.923} C_VEL
LIN {X 0,Y 573.253,Z 248.705,A -85,B 0,C 180,E1 -2052.988,E2 -2052.988} C_VEL
LIN {X 0,Y 573.263,Z 248.704,A -85,B 0,C 180,E1 -2055.806,E2 -2055.806} C_VEL
LIN {X 0,Y 573.273,Z 248.704,A -85,B 0,C 180,E1 -2058.733,E2 -2058.733} C_VEL
LIN {X 0,Y 573.3,Z 248.7,A -85,B 0,C 180,E1 -2061.54,E2 -2061.54} C_VEL
LIN {X 0,Y 573.286,Z 248.7,A -85,B 0,C 180,E1 -2064.371,E2 -2064.371} C_VEL
LIN {X 0,Y 573.154,Z 248.721,A -85,B 0,C 180,E1 -2065.78,E2 -2065.78} C_VEL
LIN {X 0,Y 573.141,Z 251.309,A -85,B 0,C 180,E1 -2068.594,E2 -2068.594} C_VEL
LIN {X 0,Y 573.111,Z 254.131,A -85,B 0,C 180,E1 -2071.405,E2 -2071.405} C_VEL
LIN {X 0,Y 573.023,Z 256.942,A -85,B 0,C 180,E1 -2074.22,E2 -2074.22} C_VEL
LIN {X 0,Y 573.02,Z 259.754,A -85,B 0,C 180,E1 -2077.044,E2 -2077.044} C_VEL
LIN {X 0,Y 572.961,Z 262.851,A -85,B 0,C 180,E1 -2079.888,E2 -2079.888} C_VEL
LIN {X 0,Y 572.937,Z 266.184,A -85,B 0,C 180,E1 -2082.755,E2 -2082.755} C_VEL
LIN {X 0,Y 572.94,Z 269.372,A -85,B 0,C 180,E1 -2085.45,E2 -2085.45} C_VEL
LIN {X 0,Y 574.703,Z 277.493,A -85,B 0,C 180,E1 -2085.652,E2 -2085.652} C_VEL
LIN {X 0,Y 574.56,Z 292.523,A -85,B 0,C 180,E1 -2085.997,E2 -2085.997} C_VEL
LIN {X 0,Y 574.352,Z 307.343,A -85,B 0,C 180,E1 -2086.482,E2 -2086.482} C_VEL
LIN {X 0,Y 574.19,Z 321.257,A -85,B 0,C 180,E1 -2087.082,E2 -2087.082} C_VEL
LIN {X 0,Y 574.021,Z 334.931,A -85,B 0,C 180,E1 -2087.823,E2 -2087.823} C_VEL
LIN {X 0,Y 573.841,Z 347.597,A -85,B 0,C 180,E1 -2088.66,E2 -2088.66} C_VEL
LIN {X 0,Y 573.625,Z 360.092,A -85,B 0,C 180,E1 -2089.652,E2 -2089.652} C_VEL
LIN {X 0,Y 573.485,Z 370.433,A -85,B 0,C 180,E1 -2090.629,E2 -2090.629} C_VEL
LIN {X 0,Y 573.321,Z 380.651,A -85,B 0,C 180,E1 -2091.765,E2 -2091.765} C_VEL
LIN {X 0,Y 573.229,Z 389.337,A -85,B 0,C 180,E1 -2092.908,E2 -2092.908} C_VEL
LIN {X 0,Y 573.155,Z 397.87,A -85,B 0,C 180,E1 -2094.253,E2 -2094.253} C_VEL
LIN {X 0,Y 573.05,Z 404.052,A -85,B 0,C 180,E1 -2095.419,E2 -2095.419} C_VEL
LIN {X 0,Y 573.047,Z 409.536,A -85,B 0,C 180,E1 -2096.69,E2 -2096.69} C_VEL
LIN {X 0,Y 572.982,Z 413.969,A -85,B 0,C 180,E1 -2097.981,E2 -2097.981} C_VEL
LIN {X 0,Y 572.962,Z 417.706,A -85,B 0,C 180,E1 -2099.44,E2 -2099.44} C_VEL
LIN {X 0,Y 572.947,Z 420.274,A -85,B 0,C 180,E1 -2101.009,E2 -2101.009} C_VEL
LIN {X 0,Y 572.94,Z 421.274,A -85,B 0,C 180,E1 -2102.181,E2 -2102.181} C_VEL
LIN {X 0,Y 572.952,Z 421.405,A -85,B 0,C 180,E1 -2103.502,E2 -2103.502} C_VEL
LIN {X 0,Y 572.954,Z 420.662,A -85,B 0,C 180,E1 -2104.733,E2 -2104.733} C_VEL
LIN {X 0,Y 572.92,Z 418.845,A -85,B 0,C 180,E1 -2106.072,E2 -2106.072} C_VEL
LIN {X 0,Y 572.953,Z 416.636,A -85,B 0,C 180,E1 -2107.128,E2 -2107.128} C_VEL
LIN {X 0,Y 572.993,Z 413.445,A -85,B 0,C 180,E1 -2108.283,E2 -2108.283} C_VEL
LIN {X 0,Y 573.045,Z 408.637,A -85,B 0,C 180,E1 -2109.623,E2 -2109.623} C_VEL
LIN {X 0,Y 573.054,Z 402.372,A -85,B 0,C 180,E1 -2111.005,E2 -2111.005} C_VEL
LIN {X 0,Y 573.135,Z 394.451,A -85,B 0,C 180,E1 -2112.409,E2 -2112.409} C_VEL
LIN {X 0,Y 573.29,Z 385.759,A -85,B 0,C 180,E1 -2113.676,E2 -2113.676} C_VEL
LIN {X 0,Y 573.396,Z 376.623,A -85,B 0,C 180,E1 -2114.798,E2 -2114.798} C_VEL
LIN {X 0,Y 573.536,Z 366.414,A -85,B 0,C 180,E1 -2115.862,E2 -2115.862} C_VEL
LIN {X 0,Y 573.746,Z 353.99,A -85,B 0,C 180,E1 -2116.945,E2 -2116.945} C_VEL
LIN {X 0,Y 573.954,Z 341.576,A -85,B 0,C 180,E1 -2117.847,E2 -2117.847} C_VEL
LIN {X 0,Y 574.151,Z 328.654,A -85,B 0,C 180,E1 -2118.626,E2 -2118.626} C_VEL
LIN {X 0,Y 574.344,Z 314.795,A -85,B 0,C 180,E1 -2119.302,E2 -2119.302} C_VEL
LIN {X 0,Y 574.505,Z 300.808,A -85,B 0,C 180,E1 -2119.836,E2 -2119.836} C_VEL
LIN {X 0,Y 574.662,Z 286.087,A -85,B 0,C 180,E1 -2120.255,E2 -2120.255} C_VEL
LIN {X 0,Y 574.54,Z 276.11,A -85,B 0,C 180,E1 -2120.47,E2 -2120.47} C_VEL
LIN {X 0,Y 572.964,Z 269.376,A -85,B 0,C 180,E1 -2120.636,E2 -2120.636} C_VEL
LIN {X 0,Y 572.956,Z 266.51,A -85,B 0,C 180,E1 -2123.057,E2 -2123.057} C_VEL
LIN {X 0,Y 572.957,Z 263.486,A -85,B 0,C 180,E1 -2125.652,E2 -2125.652} C_VEL
LIN {X 0,Y 572.993,Z 260.609,A -85,B 0,C 180,E1 -2128.171,E2 -2128.171} C_VEL
LIN {X 0,Y 573.034,Z 258.355,A -85,B 0,C 180,E1 -2130.622,E2 -2130.622} C_VEL
LIN {X 0,Y 573.044,Z 256.106,A -85,B 0,C 180,E1 -2133.015,E2 -2133.015} C_VEL
LIN {X 0,Y 573.127,Z 253.83,A -85,B 0,C 180,E1 -2135.36,E2 -2135.36} C_VEL
LIN {X 0,Y 573.101,Z 251.479,A -85,B 0,C 180,E1 -2137.658,E2 -2137.658} C_VEL
LIN {X 0,Y 573.137,Z 248.723,A -85,B 0,C 180,E1 -2140.667,E2 -2140.667} C_VEL
LIN {X 0,Y 573.254,Z 248.706,A -85,B 0,C 180,E1 -2142.99,E2 -2142.99} C_VEL
LIN {X 0,Y 573.267,Z 248.704,A -85,B 0,C 180,E1 -2145.808,E2 -2145.808} C_VEL
LIN {X 0,Y 573.256,Z 248.707,A -85,B 0,C 180,E1 -2148.746,E2 -2148.746} C_VEL
LIN {X 0,Y 573.287,Z 248.701,A -85,B 0,C 180,E1 -2151.541,E2 -2151.541} C_VEL
LIN {X 0,Y 573.289,Z 248.701,A -85,B 0,C 180,E1 -2154.373,E2 -2154.373} C_VEL
LIN {X 0,Y 573.309,Z 248.698,A -85,B 0,C 180,E1 -2157.893,E2 -2157.893} C_VEL
LIN {X 0,Y 573.329,Z 248.696,A -85,B 0,C 180,E1 -2160.703,E2 -2160.703} C_VEL
LIN {X 0,Y 573.234,Z 248.71,A -85,B 0,C 180,E1 -2163.515,E2 -2163.515} C_VEL
LIN {X 0,Y 573.29,Z 248.703,A -85,B 0,C 180,E1 -2165.629,E2 -2165.629} C_VEL
LIN {X 0,Y 573.288,Z 248.7,A -85,B 0,C 180,E1 -2168.46,E2 -2168.46} C_VEL
LIN {X 0,Y 573.268,Z 248.703,A -85,B 0,C 180,E1 -2171.313,E2 -2171.313} C_VEL
LIN {X 0,Y 573.271,Z 248.704,A -85,B 0,C 180,E1 -2174.194,E2 -2174.194} C_VEL
LIN {X 0,Y 573.255,Z 248.706,A -85,B 0,C 180,E1 -2177.112,E2 -2177.112} C_VEL
LIN {X 0,Y 573.254,Z 248.705,A -85,B 0,C 180,E1 -2180.077,E2 -2180.077} C_VEL
LIN {X 0,Y 573.236,Z 248.708,A -85,B 0,C 180,E1 -2182.338,E2 -2182.338} C_VEL
LIN {X 0,Y 573.256,Z 248.705,A -85,B 0,C 180,E1 -2185.41,E2 -2185.41} C_VEL
LIN {X 0,Y 573.251,Z 248.707,A -85,B 0,C 180,E1 -2188.03,E2 -2188.03} C_VEL
LIN {X 0,Y 573.244,Z 248.707,A -85,B 0,C 180,E1 -2190.177,E2 -2190.177} C_VEL
LIN {X 0,Y 573.251,Z 248.706,A -85,B 0,C 180,E1 -2192.646,E2 -2192.646} C_VEL
LIN {X 0,Y 573.207,Z 248.715,A -85,B 0,C 180,E1 -2195.188,E2 -2195.188} C_VEL
LIN {X 0,Y 573.234,Z 248.709,A -85,B 0,C 180,E1 -2197.808,E2 -2197.808} C_VEL
LIN {X 0,Y 573.268,Z 248.706,A -85,B 0,C 180,E1 -2200.529,E2 -2200.529} C_VEL
LIN {X 0,Y 573.242,Z 248.709,A -85,B 0,C 180,E1 -2203.67,E2 -2203.67} C_VEL
LIN {X 0,Y 573.246,Z 248.708,A -85,B 0,C 180,E1 -2206.642,E2 -2206.642} C_VEL
LIN {X 0,Y 573.285,Z 248.845,A -85,B 0,C 180,E1 -2207.094,E2 -2207.094} C_VEL
LIN {X 0,Y 573.853,Z 252.635,A -85,B 0,C 180,E1 -2208.599,E2 -2208.599} C_VEL
LIN {X 0,Y 573.845,Z 259.123,A -85,B 0,C 180,E1 -2210.922,E2 -2210.922} C_VEL
LIN {X 0,Y 573.748,Z 266.499,A -85,B 0,C 180,E1 -2213.553,E2 -2213.553} C_VEL
LIN {X 0,Y 573.611,Z 275.162,A -85,B 0,C 180,E1 -2216.541,E2 -2216.541} C_VEL
LIN {X 0,Y 573.507,Z 282.733,A -85,B 0,C 180,E1 -2219.072,E2 -2219.072} C_VEL
LIN {X 0,Y 573.457,Z 290.016,A -85,B 0,C 180,E1 -2221.448,E2 -2221.448} C_VEL
LIN {X 0,Y 573.389,Z 298.68,A -85,B 0,C 180,E1 -2224.208,E2 -2224.208} C_VEL
LIN {X 0,Y 573.255,Z 307.345,A -85,B 0,C 180,E1 -2226.902,E2 -2226.902} C_VEL
LIN {X 0,Y 573.216,Z 316.01,A -85,B 0,C 180,E1 -2229.548,E2 -2229.548} C_VEL
LIN {X 0,Y 573.163,Z 325.427,A -85,B 0,C 180,E1 -2232.374,E2 -2232.374} C_VEL
LIN {X 0,Y 574.715,Z 332.409,A -85,B 0,C 180,E1 -2232.523,E2 -2232.523} C_VEL
LIN {X 0,Y 574.634,Z 347.925,A -85,B 0,C 180,E1 -2232.835,E2 -2232.835} C_VEL
LIN {X 0,Y 574.498,Z 363.221,A -85,B 0,C 180,E1 -2233.293,E2 -2233.293} C_VEL
LIN {X 0,Y 574.281,Z 376.837,A -85,B 0,C 180,E1 -2233.835,E2 -2233.835} C_VEL
LIN {X 0,Y 574.08,Z 391.114,A -85,B 0,C 180,E1 -2234.558,E2 -2234.558} C_VEL
LIN {X 0,Y 573.887,Z 404.711,A -85,B 0,C 180,E1 -2235.412,E2 -2235.412} C_VEL
LIN {X 0,Y 573.689,Z 417.173,A -85,B 0,C 180,E1 -2236.36,E2 -2236.36} C_VEL
LIN {X 0,Y 573.511,Z 428.978,A -85,B 0,C 180,E1 -2237.437,E2 -2237.437} C_VEL
LIN {X 0,Y 573.349,Z 438.905,A -85,B 0,C 180,E1 -2238.511,E2 -2238.511} C_VEL
LIN {X 0,Y 573.256,Z 448.621,A -85,B 0,C 180,E1 -2239.761,E2 -2239.761} C_VEL
LIN {X 0,Y 573.135,Z 456.723,A -85,B 0,C 180,E1 -2241.006,E2 -2241.006} C_VEL
LIN {X 0,Y 573.093,Z 463.428,A -85,B 0,C 180,E1 -2242.248,E2 -2242.248} C_VEL
LIN {X 0,Y 573.015,Z 469.609,A -85,B 0,C 180,E1 -2243.663,E2 -2243.663} C_VEL
LIN {X 0,Y 572.951,Z 474.385,A -85,B 0,C 180,E1 -2245.075,E2 -2245.075} C_VEL
LIN {X 0,Y 573.005,Z 477.888,A -85,B 0,C 180,E1 -2246.485,E2 -2246.485} C_VEL
LIN {X 0,Y 572.938,Z 480.194,A -85,B 0,C 180,E1 -2247.892,E2 -2247.892} C_VEL
LIN {X 0,Y 572.936,Z 481.35,A -85,B 0,C 180,E1 -2249.298,E2 -2249.298} C_VEL
LIN {X 0,Y 572.936,Z 481.349,A -85,B 0,C 180,E1 -2250.703,E2 -2250.703} C_VEL
LIN {X 0,Y 572.938,Z 480.192,A -85,B 0,C 180,E1 -2252.109,E2 -2252.109} C_VEL
LIN {X 0,Y 573.005,Z 477.885,A -85,B 0,C 180,E1 -2253.516,E2 -2253.516} C_VEL
LIN {X 0,Y 572.951,Z 474.383,A -85,B 0,C 180,E1 -2254.926,E2 -2254.926} C_VEL
LIN {X 0,Y 573.014,Z 469.606,A -85,B 0,C 180,E1 -2256.338,E2 -2256.338} C_VEL
LIN {X 0,Y 573.094,Z 463.422,A -85,B 0,C 180,E1 -2257.753,E2 -2257.753} C_VEL
LIN {X 0,Y 573.136,Z 455.648,A -85,B 0,C 180,E1 -2259.173,E2 -2259.173} C_VEL
LIN {X 0,Y 573.27,Z 447.366,A -85,B 0,C 180,E1 -2260.418,E2 -2260.418} C_VEL
LIN {X 0,Y 573.387,Z 437.387,A -85,B 0,C 180,E1 -2261.668,E2 -2261.668} C_VEL
LIN {X 0,Y 573.568,Z 427.186,A -85,B 0,C 180,E1 -2262.742,E2 -2262.742} C_VEL
LIN {X 0,Y 573.725,Z 415.011,A -85,B 0,C 180,E1 -2263.82,E2 -2263.82} C_VEL
LIN {X 0,Y 573.963,Z 401.89,A -85,B 0,C 180,E1 -2264.781,E2 -2264.781} C_VEL
LIN {X 0,Y 574.075,Z 389.515,A -85,B 0,C 180,E1 -2265.534,E2 -2265.534} C_VEL
LIN {X 0,Y 574.302,Z 374.829,A -85,B 0,C 180,E1 -2266.257,E2 -2266.257} C_VEL
LIN {X 0,Y 574.511,Z 360.604,A -85,B 0,C 180,E1 -2266.799,E2 -2266.799} C_VEL
LIN {X 0,Y 574.683,Z 345.918,A -85,B 0,C 180,E1 -2267.214,E2 -2267.214} C_VEL
LIN {X 0,Y 574.602,Z 331.817,A -85,B 0,C 180,E1 -2267.49,E2 -2267.49} C_VEL
LIN {X 0,Y 573.169,Z 325.371,A -85,B 0,C 180,E1 -2267.643,E2 -2267.643} C_VEL
LIN {X 0,Y 573.21,Z 316.006,A -85,B 0,C 180,E1 -2270.453,E2 -2270.453} C_VEL
LIN {X 0,Y 573.277,Z 307.16,A -85,B 0,C 180,E1 -2273.154,E2 -2273.154} C_VEL
LIN {X 0,Y 573.391,Z 298.677,A -85,B 0,C 180,E1 -2275.793,E2 -2275.793} C_VEL
LIN {X 0,Y 573.459,Z 290.012,A -85,B 0,C 180,E1 -2278.553,E2 -2278.553} C_VEL
LIN {X 0,Y 573.556,Z 281.348,A -85,B 0,C 180,E1 -2281.384,E2 -2281.384} C_VEL
LIN {X 0,Y 573.63,Z 272.683,A -85,B 0,C 180,E1 -2284.304,E2 -2284.304} C_VEL
LIN {X 0,Y 573.785,Z 264.264,A -85,B 0,C 180,E1 -2287.236,E2 -2287.236} C_VEL
LIN {X 0,Y 573.869,Z 256.457,A -85,B 0,C 180,E1 -2290.013,E2 -2290.013} C_VEL
